LIN {X 0,Y 417.827,Z 989.103,A -85,B 0,C 180,E1 9549.226,E2 9549.226} C_VEL
LIN {X 0,Y 425.019,Z 968.051,A -85,B 0,C 180,E1 9548.696,E2 9548.696} C_VEL
LIN {X 0,Y 431.28,Z 946.58,A -85,B 0,C 180,E1 9548.255,E2 9548.255} C_VEL
LIN {X 0,Y 437.071,Z 922.468,A -85,B 0,C 180,E1 9547.851,E2 9547.851} C_VEL
LIN {X 0,Y 442.216,Z 893.072,A -85,B 0,C 180,E1 9547.412,E2 9547.412} C_VEL
LIN {X 0,Y 449.934,Z 826.101,A -85,B 0,C 180,E1 9546.506,E2 9546.506} C_VEL
LIN {X 0,Y 462.128,Z 717.477,A -85,B 0,C 180,E1 9545.058,E2 9545.058} C_VEL
LIN {X 0,Y 461.175,Z 715.537,A -85,B 0,C 180,E1 9543.107,E2 9543.107} C_VEL
LIN {X 0,Y 460.734,Z 712.812,A -85,B 0,C 180,E1 9540.249,E2 9540.249} C_VEL
LIN {X 0,Y 460.752,Z 712.952,A -85,B 0,C 180,E1 9538.881,E2 9538.881} C_VEL
LIN {X 0,Y 462.07,Z 717.316,A -85,B 0,C 180,E1 9534.54,E2 9534.54} C_VEL
LIN {X 0,Y 442.815,Z 887.011,A -85,B 0,C 180,E1 9532.28,E2 9532.28} C_VEL
LIN {X 0,Y 438.536,Z 912.989,A -85,B 0,C 180,E1 9531.901,E2 9531.901} C_VEL
LIN {X 0,Y 432.21,Z 940.386,A -85,B 0,C 180,E1 9531.4,E2 9531.4} C_VEL
LIN {X 0,Y 425.994,Z 962.099,A -85,B 0,C 180,E1 9530.901,E2 9530.901} C_VEL
LIN {X 0,Y 419.318,Z 981.985,A -85,B 0,C 180,E1 9530.35,E2 9530.35} C_VEL
LIN {X 0,Y 411.3,Z 1002.768,A -85,B 0,C 180,E1 9529.662,E2 9529.662} C_VEL
LIN {X 0,Y 400.652,Z 1026.921,A -85,B 0,C 180,E1 9528.701,E2 9528.701} C_VEL
LIN {X 0,Y 388.49,Z 1050.508,A -85,B 0,C 180,E1 9527.54,E2 9527.54} C_VEL
LIN {X 0,Y 377.454,Z 1069.69,A -85,B 0,C 180,E1 9526.414,E2 9526.414} C_VEL
LIN {X 0,Y 366.103,Z 1087.649,A -85,B 0,C 180,E1 9525.162,E2 9525.162} C_VEL
LIN {X 0,Y 352.977,Z 1106.617,A -85,B 0,C 180,E1 9523.599,E2 9523.599} C_VEL
LIN {X 0,Y 336.444,Z 1128.11,A -85,B 0,C 180,E1 9521.416,E2 9521.416} C_VEL
LIN {X 0,Y 323.396,Z 1143.609,A -85,B 0,C 180,E1 9519.493,E2 9519.493} C_VEL
LIN {X 0,Y 309.958,Z 1158.478,A -85,B 0,C 180,E1 9517.28,E2 9517.28} C_VEL
LIN {X 0,Y 296.26,Z 1172.662,A -85,B 0,C 180,E1 9514.73,E2 9514.73} C_VEL
LIN {X 0,Y 279.66,Z 1188.763,A -85,B 0,C 180,E1 9511.134,E2 9511.134} C_VEL
LIN {X 0,Y 264.844,Z 1202.074,A -85,B 0,C 180,E1 9507.319,E2 9507.319} C_VEL
LIN {X 0,Y 252.417,Z 1212.779,A -85,B 0,C 180,E1 9503.505,E2 9503.505} C_VEL
LIN {X 0,Y 241.138,Z 1222.219,A -85,B 0,C 180,E1 9499.339,E2 9499.339} C_VEL
LIN {X 0,Y 228.776,Z 1232.449,A -85,B 0,C 180,E1 9493.655,E2 9493.655} C_VEL
LIN {X 0,Y 218.042,Z 1241.237,A -85,B 0,C 180,E1 9487.067,E2 9487.067} C_VEL
LIN {X 0,Y 211.235,Z 1247.103,A -85,B 0,C 180,E1 9481.362,E2 9481.362} C_VEL
LIN {X 0,Y 206.073,Z 1251.951,A -85,B 0,C 180,E1 9475.261,E2 9475.261} C_VEL
LIN {X 0,Y 202.665,Z 1255.674,A -85,B 0,C 180,E1 9468.989,E2 9468.989} C_VEL
LIN {X 0,Y 200.676,Z 1258.635,A -85,B 0,C 180,E1 9461.774,E2 9461.774} C_VEL
LIN {X 0,Y 200.109,Z 1260.066,A -85,B 0,C 180,E1 9455.147,E2 9455.147} C_VEL
LIN {X 0,Y 200.012,Z 1260.414,A -85,B 0,C 180,E1 9449.414,E2 9449.414} C_VEL
LIN {X 0,Y 200.159,Z 1259.917,A -85,B 0,C 180,E1 9443.678,E2 9443.678} C_VEL
LIN {X 0,Y 200.883,Z 1258.243,A -85,B 0,C 180,E1 9437.044,E2 9437.044} C_VEL
LIN {X 0,Y 202.764,Z 1255.578,A -85,B 0,C 180,E1 9430.695,E2 9430.695} C_VEL
LIN {X 0,Y 206.041,Z 1252.022,A -85,B 0,C 180,E1 9424.707,E2 9424.707} C_VEL
LIN {X 0,Y 210.915,Z 1247.435,A -85,B 0,C 180,E1 9418.874,E2 9418.874} C_VEL
LIN {X 0,Y 217.804,Z 1241.484,A -85,B 0,C 180,E1 9413.016,E2 9413.016} C_VEL
LIN {X 0,Y 228.254,Z 1232.955,A -85,B 0,C 180,E1 9406.535,E2 9406.535} C_VEL
LIN {X 0,Y 240.93,Z 1222.476,A -85,B 0,C 180,E1 9400.66,E2 9400.66} C_VEL
LIN {X 0,Y 252.341,Z 1212.937,A -85,B 0,C 180,E1 9396.437,E2 9396.437} C_VEL
LIN {X 0,Y 264.769,Z 1202.248,A -85,B 0,C 180,E1 9392.619,E2 9392.619} C_VEL
LIN {X 0,Y 280.29,Z 1188.333,A -85,B 0,C 180,E1 9388.637,E2 9388.637} C_VEL
LIN {X 0,Y 296.47,Z 1172.615,A -85,B 0,C 180,E1 9385.148,E2 9385.148} C_VEL
LIN {X 0,Y 309.897,Z 1158.729,A -85,B 0,C 180,E1 9382.649,E2 9382.649} C_VEL
LIN {X 0,Y 323.344,Z 1143.878,A -85,B 0,C 180,E1 9380.436,E2 9380.436} C_VEL
LIN {X 0,Y 338.051,Z 1126.397,A -85,B 0,C 180,E1 9378.28,E2 9378.28} C_VEL
LIN {X 0,Y 354.452,Z 1104.814,A -85,B 0,C 180,E1 9376.136,E2 9376.136} C_VEL
LIN {X 0,Y 366.727,Z 1087.025,A -85,B 0,C 180,E1 9374.689,E2 9374.689} C_VEL
LIN {X 0,Y 377.843,Z 1069.412,A -85,B 0,C 180,E1 9373.467,E2 9373.467} C_VEL
LIN {X 0,Y 388.96,Z 1050.061,A -85,B 0,C 180,E1 9372.335,E2 9372.335} C_VEL
LIN {X 0,Y 401.541,Z 1025.448,A -85,B 0,C 180,E1 9371.137,E2 9371.137} C_VEL
LIN {X 0,Y 411.533,Z 1002.753,A -85,B 0,C 180,E1 9370.241,E2 9370.241} C_VEL
LIN {X 0,Y 419.451,Z 982.262,A -85,B 0,C 180,E1 9369.562,E2 9369.562} C_VEL
LIN {X 0,Y 426.457,Z 961.37,A -85,B 0,C 180,E1 9368.985,E2 9368.985} C_VEL
LIN {X 0,Y 433.115,Z 937.897,A -85,B 0,C 180,E1 9368.453,E2 9368.453} C_VEL
LIN {X 0,Y 439.471,Z 909.083,A -85,B 0,C 180,E1 9367.944,E2 9367.944} C_VEL
LIN {X 0,Y 443.203,Z 885.906,A -85,B 0,C 180,E1 9367.611,E2 9367.611} C_VEL
LIN {X 0,Y 461.965,Z 720.462,A -85,B 0,C 180,E1 9365.408,E2 9365.408} C_VEL
LIN {X 0,Y 462.048,Z 718.822,A -85,B 0,C 180,E1 9365.242,E2 9365.242} C_VEL
LIN {X 0,Y 461.875,Z 718.154,A -85,B 0,C 180,E1 9364.869,E2 9364.869} C_VEL
LIN {X 0,Y 461.404,Z 718.961,A -85,B 0,C 180,E1 9364.262,E2 9364.262} C_VEL
LIN {X 0,Y 460.384,Z 722.397,A -85,B 0,C 180,E1 9363.028,E2 9363.028} C_VEL
LIN {X 0,Y 460.143,Z 722.68,A -85,B 0,C 180,E1 9362.446,E2 9362.446} C_VEL
LIN {X 0,Y 460.028,Z 720.774,A -85,B 0,C 180,E1 9360.374,E2 9360.374} C_VEL
LIN {X 0,Y 460.024,Z 721.081,A -85,B 0,C 180,E1 9359.502,E2 9359.502} C_VEL
LIN {X 0,Y 460.881,Z 724.724,A -85,B 0,C 180,E1 9355.84,E2 9355.84} C_VEL
LIN {X 0,Y 441.798,Z 890.537,A -85,B 0,C 180,E1 9353.66,E2 9353.66} C_VEL
LIN {X 0,Y 437.471,Z 916.586,A -85,B 0,C 180,E1 9353.287,E2 9353.287} C_VEL
LIN {X 0,Y 430.938,Z 944.462,A -85,B 0,C 180,E1 9352.846,E2 9352.846} C_VEL
LIN {X 0,Y 424.579,Z 966.3,A -85,B 0,C 180,E1 9352.422,E2 9352.422} C_VEL
LIN {X 0,Y 417.486,Z 987.052,A -85,B 0,C 180,E1 9351.926,E2 9351.926} C_VEL
LIN {X 0,Y 409.171,Z 1008.194,A -85,B 0,C 180,E1 9351.313,E2 9351.313} C_VEL
LIN {X 0,Y 397.239,Z 1034.481,A -85,B 0,C 180,E1 9350.363,E2 9350.363} C_VEL
LIN {X 0,Y 385.977,Z 1055.977,A -85,B 0,C 180,E1 9349.401,E2 9349.401} C_VEL
LIN {X 0,Y 375.148,Z 1074.641,A -85,B 0,C 180,E1 9348.398,E2 9348.398} C_VEL
LIN {X 0,Y 363.473,Z 1092.965,A -85,B 0,C 180,E1 9347.232,E2 9347.232} C_VEL
LIN {X 0,Y 350.354,Z 1111.817,A -85,B 0,C 180,E1 9345.792,E2 9345.792} C_VEL
LIN {X 0,Y 332.937,Z 1134.393,A -85,B 0,C 180,E1 9343.661,E2 9343.661} C_VEL
LIN {X 0,Y 318.986,Z 1150.867,A -85,B 0,C 180,E1 9341.732,E2 9341.732} C_VEL
LIN {X 0,Y 305.166,Z 1166.066,A -85,B 0,C 180,E1 9339.584,E2 9339.584} C_VEL
LIN {X 0,Y 290.981,Z 1180.683,A -85,B 0,C 180,E1 9337.076,E2 9337.076} C_VEL
LIN {X 0,Y 273.041,Z 1197.971,A -85,B 0,C 180,E1 9333.336,E2 9333.336} C_VEL
LIN {X 0,Y 258.369,Z 1211.155,A -85,B 0,C 180,E1 9329.671,E2 9329.671} C_VEL
LIN {X 0,Y 245.406,Z 1222.365,A -85,B 0,C 180,E1 9325.787,E2 9325.787} C_VEL
LIN {X 0,Y 233.12,Z 1232.701,A -85,B 0,C 180,E1 9321.332,E2 9321.332} C_VEL
LIN {X 0,Y 219.784,Z 1243.853,A -85,B 0,C 180,E1 9315.157,E2 9315.157} C_VEL
LIN {X 0,Y 209.458,Z 1252.521,A -85,B 0,C 180,E1 9308.721,E2 9308.721} C_VEL
LIN {X 0,Y 202.639,Z 1258.658,A -85,B 0,C 180,E1 9302.886,E2 9302.886} C_VEL
LIN {X 0,Y 197.807,Z 1263.476,A -85,B 0,C 180,E1 9297.074,E2 9297.074} C_VEL
LIN {X 0,Y 194.579,Z 1267.316,A -85,B 0,C 180,E1 9291.096,E2 9291.096} C_VEL
LIN {X 0,Y 192.761,Z 1270.194,A -85,B 0,C 180,E1 9285.045,E2 9285.045} C_VEL
LIN {X 0,Y 192.092,Z 1271.973,A -85,B 0,C 180,E1 9279.602,E2 9279.602} C_VEL
LIN {X 0,Y 192.021,Z 1272.964,A -85,B 0,C 180,E1 9274.493,E2 9274.493} C_VEL
LIN {X 0,Y 192.011,Z 1273.253,A -85,B 0,C 180,E1 9269.119,E2 9269.119} C_VEL
LIN {X 0,Y 192.03,Z 1272.694,A -85,B 0,C 180,E1 9263.436,E2 9263.436} C_VEL
LIN {X 0,Y 192.495,Z 1270.789,A -85,B 0,C 180,E1 9256.497,E2 9256.497} C_VEL
LIN {X 0,Y 194.208,Z 1267.811,A -85,B 0,C 180,E1 9249.837,E2 9249.837} C_VEL
LIN {X 0,Y 197.39,Z 1263.897,A -85,B 0,C 180,E1 9243.544,E2 9243.544} C_VEL
LIN {X 0,Y 202.332,Z 1258.908,A -85,B 0,C 180,E1 9237.425,E2 9237.425} C_VEL
LIN {X 0,Y 209.057,Z 1252.815,A -85,B 0,C 180,E1 9231.573,E2 9231.573} C_VEL
LIN {X 0,Y 218.472,Z 1244.84,A -85,B 0,C 180,E1 9225.559,E2 9225.559} C_VEL
LIN {X 0,Y 232.595,Z 1233.068,A -85,B 0,C 180,E1 9218.876,E2 9218.876} C_VEL
LIN {X 0,Y 244.771,Z 1222.819,A -85,B 0,C 180,E1 9214.418,E2 9214.418} C_VEL
LIN {X 0,Y 257.409,Z 1211.888,A -85,B 0,C 180,E1 9210.588,E2 9210.588} C_VEL
LIN {X 0,Y 271.526,Z 1199.21,A -85,B 0,C 180,E1 9207.009,E2 9207.009} C_VEL
LIN {X 0,Y 290.131,Z 1181.388,A -85,B 0,C 180,E1 9203.08,E2 9203.08} C_VEL
LIN {X 0,Y 304.281,Z 1166.834,A -85,B 0,C 180,E1 9200.557,E2 9200.557} C_VEL
LIN {X 0,Y 317.858,Z 1151.944,A -85,B 0,C 180,E1 9198.427,E2 9198.427} C_VEL
LIN {X 0,Y 330.96,Z 1136.545,A -85,B 0,C 180,E1 9196.587,E2 9196.587} C_VEL
LIN {X 0,Y 345.571,Z 1118.021,A -85,B 0,C 180,E1 9194.751,E2 9194.751} C_VEL
LIN {X 0,Y 361.758,Z 1095.238,A -85,B 0,C 180,E1 9192.937,E2 9192.937} C_VEL
LIN {X 0,Y 374.151,Z 1075.917,A -85,B 0,C 180,E1 9191.688,E2 9191.688} C_VEL
LIN {X 0,Y 385.049,Z 1057.238,A -85,B 0,C 180,E1 9190.671,E2 9190.671} C_VEL
LIN {X 0,Y 396.029,Z 1036.414,A -85,B 0,C 180,E1 9189.725,E2 9189.725} C_VEL
LIN {X 0,Y 408.494,Z 1009.289,A -85,B 0,C 180,E1 9188.729,E2 9188.729} C_VEL
LIN {X 0,Y 417.04,Z 987.634,A -85,B 0,C 180,E1 9188.096,E2 9188.096} C_VEL
LIN {X 0,Y 424.156,Z 966.885,A -85,B 0,C 180,E1 9187.597,E2 9187.597} C_VEL
LIN {X 0,Y 430.377,Z 945.642,A -85,B 0,C 180,E1 9187.18,E2 9187.18} C_VEL
LIN {X 0,Y 436.755,Z 919.053,A -85,B 0,C 180,E1 9186.754,E2 9186.754} C_VEL
LIN {X 0,Y 441.451,Z 891.288,A -85,B 0,C 180,E1 9186.354,E2 9186.354} C_VEL
LIN {X 0,Y 454.023,Z 782.367,A -85,B 0,C 180,E1 9184.916,E2 9184.916} C_VEL
LIN {X 0,Y 460.65,Z 724.372,A -85,B 0,C 180,E1 9184.139,E2 9184.139} C_VEL
LIN {X 0,Y 459.759,Z 720.752,A -85,B 0,C 180,E1 9180.249,E2 9180.249} C_VEL
LIN {X 0,Y 459.767,Z 720.977,A -85,B 0,C 180,E1 9178.878,E2 9178.878} C_VEL
LIN {X 0,Y 460.589,Z 724.432,A -85,B 0,C 180,E1 9175.442,E2 9175.442} C_VEL
LIN {X 0,Y 441.811,Z 887.296,A -85,B 0,C 180,E1 9173.309,E2 9173.309} C_VEL
LIN {X 0,Y 437.45,Z 913.431,A -85,B 0,C 180,E1 9172.937,E2 9172.937} C_VEL
LIN {X 0,Y 431.084,Z 940.66,A -85,B 0,C 180,E1 9172.454,E2 9172.454} C_VEL
LIN {X 0,Y 424.797,Z 962.372,A -85,B 0,C 180,E1 9171.971,E2 9171.971} C_VEL
LIN {X 0,Y 418.044,Z 982.258,A -85,B 0,C 180,E1 9171.437,E2 9171.437} C_VEL
LIN {X 0,Y 410.172,Z 1002.448,A -85,B 0,C 180,E1 9170.791,E2 9170.791} C_VEL
LIN {X 0,Y 399.603,Z 1026.198,A -85,B 0,C 180,E1 9169.881,E2 9169.881} C_VEL
LIN {X 0,Y 387.316,Z 1049.895,A -85,B 0,C 180,E1 9168.762,E2 9168.762} C_VEL
LIN {X 0,Y 376.073,Z 1069.234,A -85,B 0,C 180,E1 9167.665,E2 9167.665} C_VEL
LIN {X 0,Y 364.98,Z 1086.599,A -85,B 0,C 180,E1 9166.499,E2 9166.499} C_VEL
LIN {X 0,Y 352.723,Z 1104.142,A -85,B 0,C 180,E1 9165.121,E2 9165.121} C_VEL
LIN {X 0,Y 336.944,Z 1124.789,A -85,B 0,C 180,E1 9163.157,E2 9163.157} C_VEL
LIN {X 0,Y 320.707,Z 1143.762,A -85,B 0,C 180,E1 9160.891,E2 9160.891} C_VEL
LIN {X 0,Y 307.656,Z 1157.92,A -85,B 0,C 180,E1 9158.836,E2 9158.836} C_VEL
LIN {X 0,Y 294.353,Z 1171.42,A -85,B 0,C 180,E1 9156.485,E2 9156.485} C_VEL
LIN {X 0,Y 280.096,Z 1184.997,A -85,B 0,C 180,E1 9153.612,E2 9153.612} C_VEL
LIN {X 0,Y 262.461,Z 1200.665,A -85,B 0,C 180,E1 9149.402,E2 9149.402} C_VEL
LIN {X 0,Y 248.783,Z 1212.049,A -85,B 0,C 180,E1 9145.456,E2 9145.456} C_VEL
LIN {X 0,Y 236.897,Z 1221.601,A -85,B 0,C 180,E1 9141.316,E2 9141.316} C_VEL
LIN {X 0,Y 225.735,Z 1230.361,A -85,B 0,C 180,E1 9136.568,E2 9136.568} C_VEL
LIN {X 0,Y 214.002,Z 1239.604,A -85,B 0,C 180,E1 9130.131,E2 9130.131} C_VEL
LIN {X 0,Y 204.797,Z 1246.886,A -85,B 0,C 180,E1 9123.132,E2 9123.132} C_VEL
LIN {X 0,Y 199.289,Z 1251.628,A -85,B 0,C 180,E1 9117.15,E2 9117.15} C_VEL
LIN {X 0,Y 195.512,Z 1255.333,A -85,B 0,C 180,E1 9110.961,E2 9110.961} C_VEL
LIN {X 0,Y 193.263,Z 1258.045,A -85,B 0,C 180,E1 9104.65,E2 9104.65} C_VEL
LIN {X 0,Y 192.325,Z 1259.643,A -85,B 0,C 180,E1 9098.957,E2 9098.957} C_VEL
LIN {X 0,Y 192.078,Z 1260.431,A -85,B 0,C 180,E1 9093.866,E2 9093.866} C_VEL
LIN {X 0,Y 192.041,Z 1260.588,A -85,B 0,C 180,E1 9088.196,E2 9088.196} C_VEL
LIN {X 0,Y 192.229,Z 1259.986,A -85,B 0,C 180,E1 9082.515,E2 9082.515} C_VEL
LIN {X 0,Y 193.113,Z 1258.293,A -85,B 0,C 180,E1 9075.902,E2 9075.902} C_VEL
LIN {X 0,Y 195.206,Z 1255.694,A -85,B 0,C 180,E1 9069.603,E2 9069.603} C_VEL
LIN {X 0,Y 198.826,Z 1252.094,A -85,B 0,C 180,E1 9063.399,E2 9063.399} C_VEL
LIN {X 0,Y 204.155,Z 1247.461,A -85,B 0,C 180,E1 9057.389,E2 9057.389} C_VEL
LIN {X 0,Y 211.593,Z 1241.465,A -85,B 0,C 180,E1 9051.395,E2 9051.395} C_VEL
LIN {X 0,Y 223.228,Z 1232.464,A -85,B 0,C 180,E1 9044.573,E2 9044.573} C_VEL
LIN {X 0,Y 235.705,Z 1222.638,A -85,B 0,C 180,E1 9039.063,E2 9039.063} C_VEL
LIN {X 0,Y 247.471,Z 1213.209,A -85,B 0,C 180,E1 9034.881,E2 9034.881} C_VEL
LIN {X 0,Y 260.366,Z 1202.52,A -85,B 0,C 180,E1 9031.072,E2 9031.072} C_VEL
LIN {X 0,Y 276.441,Z 1188.567,A -85,B 0,C 180,E1 9027.113,E2 9027.113} C_VEL
LIN {X 0,Y 292.76,Z 1173.164,A -85,B 0,C 180,E1 9023.734,E2 9023.734} C_VEL
LIN {X 0,Y 306.964,Z 1158.832,A -85,B 0,C 180,E1 9021.197,E2 9021.197} C_VEL
LIN {X 0,Y 320.554,Z 1144.146,A -85,B 0,C 180,E1 9019.052,E2 9019.052} C_VEL
LIN {X 0,Y 335.56,Z 1126.664,A -85,B 0,C 180,E1 9016.945,E2 9016.945} C_VEL
LIN {X 0,Y 352.261,Z 1105.079,A -85,B 0,C 180,E1 9014.855,E2 9014.855} C_VEL
LIN {X 0,Y 364.365,Z 1087.854,A -85,B 0,C 180,E1 9013.489,E2 9013.489} C_VEL
LIN {X 0,Y 375.704,Z 1070.206,A -85,B 0,C 180,E1 9012.293,E2 9012.293} C_VEL
LIN {X 0,Y 386.898,Z 1051.047,A -85,B 0,C 180,E1 9011.199,E2 9011.199} C_VEL
LIN {X 0,Y 399.143,Z 1027.673,A -85,B 0,C 180,E1 9010.083,E2 9010.083} C_VEL
LIN {X 0,Y 410.175,Z 1003.011,A -85,B 0,C 180,E1 9009.132,E2 9009.132} C_VEL
LIN {X 0,Y 418.052,Z 982.895,A -85,B 0,C 180,E1 9008.486,E2 9008.486} C_VEL
LIN {X 0,Y 425.043,Z 962.361,A -85,B 0,C 180,E1 9007.934,E2 9007.934} C_VEL
LIN {X 0,Y 431.436,Z 940.255,A -85,B 0,C 180,E1 9007.442,E2 9007.442} C_VEL
LIN {X 0,Y 437.93,Z 912.126,A -85,B 0,C 180,E1 9006.948,E2 9006.948} C_VEL
LIN {X 0,Y 442.084,Z 887.108,A -85,B 0,C 180,E1 9006.595,E2 9006.595} C_VEL
LIN {X 0,Y 460.841,Z 724.411,A -85,B 0,C 180,E1 9004.449,E2 9004.449} C_VEL
LIN {X 0,Y 460.143,Z 722.68,A -85,B 0,C 180,E1 9002.446,E2 9002.446} C_VEL
LIN {X 0,Y 459.896,Z 722.863,A -85,B 0,C 180,E1 9001.548,E2 9001.548} C_VEL
LIN {X 0,Y 459.438,Z 725.568,A -85,B 0,C 180,E1 9000.265,E2 9000.265} C_VEL
LIN {X 0,Y 459.096,Z 730.018,A -85,B 0,C 180,E1 8998.499,E2 8998.499} C_VEL
LIN {X 0,Y 459.139,Z 730.581,A -85,B 0,C 180,E1 8998.079,E2 8998.079} C_VEL
LIN {X 0,Y 459.5,Z 731.895,A -85,B 0,C 180,E1 8996.745,E2 8996.745} C_VEL
LIN {X 0,Y 440.967,Z 890.402,A -85,B 0,C 180,E1 8994.699,E2 8994.699} C_VEL
LIN {X 0,Y 436.485,Z 916.989,A -85,B 0,C 180,E1 8994.327,E2 8994.327} C_VEL
LIN {X 0,Y 429.907,Z 944.576,A -85,B 0,C 180,E1 8993.905,E2 8993.905} C_VEL
LIN {X 0,Y 423.688,Z 965.735,A -85,B 0,C 180,E1 8993.511,E2 8993.511} C_VEL
LIN {X 0,Y 416.548,Z 986.465,A -85,B 0,C 180,E1 8993.037,E2 8993.037} C_VEL
LIN {X 0,Y 408.159,Z 1007.61,A -85,B 0,C 180,E1 8992.45,E2 8992.45} C_VEL
LIN {X 0,Y 396.28,Z 1033.592,A -85,B 0,C 180,E1 8991.551,E2 8991.551} C_VEL
LIN {X 0,Y 384.638,Z 1055.568,A -85,B 0,C 180,E1 8990.607,E2 8990.607} C_VEL
LIN {X 0,Y 373.581,Z 1074.375,A -85,B 0,C 180,E1 8989.633,E2 8989.633} C_VEL
LIN {X 0,Y 361.975,Z 1092.352,A -85,B 0,C 180,E1 8988.528,E2 8988.528} C_VEL
LIN {X 0,Y 349.171,Z 1110.504,A -85,B 0,C 180,E1 8987.195,E2 8987.195} C_VEL
LIN {X 0,Y 332.606,Z 1131.868,A -85,B 0,C 180,E1 8985.28,E2 8985.28} C_VEL
LIN {X 0,Y 316.811,Z 1150.212,A -85,B 0,C 180,E1 8983.218,E2 8983.218} C_VEL
LIN {X 0,Y 303.164,Z 1164.936,A -85,B 0,C 180,E1 8981.204,E2 8981.204} C_VEL
LIN {X 0,Y 289.398,Z 1178.844,A -85,B 0,C 180,E1 8978.903,E2 8978.903} C_VEL
LIN {X 0,Y 274.618,Z 1192.874,A -85,B 0,C 180,E1 8976.065,E2 8976.065} C_VEL
LIN {X 0,Y 255.602,Z 1209.708,A -85,B 0,C 180,E1 8971.679,E2 8971.679} C_VEL
LIN {X 0,Y 241.438,Z 1221.524,A -85,B 0,C 180,E1 8967.67,E2 8967.67} C_VEL
LIN {X 0,Y 229.094,Z 1231.483,A -85,B 0,C 180,E1 8963.439,E2 8963.439} C_VEL
LIN {X 0,Y 216.998,Z 1241.082,A -85,B 0,C 180,E1 8958.3,E2 8958.3} C_VEL
LIN {X 0,Y 204.163,Z 1251.305,A -85,B 0,C 180,E1 8951.03,E2 8951.03} C_VEL
LIN {X 0,Y 195.973,Z 1258.119,A -85,B 0,C 180,E1 8944.509,E2 8944.509} C_VEL
LIN {X 0,Y 190.446,Z 1263.204,A -85,B 0,C 180,E1 8938.212,E2 8938.212} C_VEL
LIN {X 0,Y 186.902,Z 1267.045,A -85,B 0,C 180,E1 8932.006,E2 8932.006} C_VEL
LIN {X 0,Y 184.877,Z 1269.927,A -85,B 0,C 180,E1 8925.699,E2 8925.699} C_VEL
LIN {X 0,Y 184.111,Z 1271.707,A -85,B 0,C 180,E1 8920.022,E2 8920.022} C_VEL
LIN {X 0,Y 184.023,Z 1272.7,A -85,B 0,C 180,E1 8914.689,E2 8914.689} C_VEL
LIN {X 0,Y 184.016,Z 1272.99,A -85,B 0,C 180,E1 8909.08,E2 8909.08} C_VEL
LIN {X 0,Y 184.032,Z 1272.502,A -85,B 0,C 180,E1 8903.463,E2 8903.463} C_VEL
LIN {X 0,Y 184.528,Z 1270.641,A -85,B 0,C 180,E1 8896.222,E2 8896.222} C_VEL
LIN {X 0,Y 186.493,Z 1267.54,A -85,B 0,C 180,E1 8888.964,E2 8888.964} C_VEL
LIN {X 0,Y 189.989,Z 1263.624,A -85,B 0,C 180,E1 8882.428,E2 8882.428} C_VEL
LIN {X 0,Y 195.332,Z 1258.633,A -85,B 0,C 180,E1 8876.103,E2 8876.103} C_VEL
LIN {X 0,Y 202.534,Z 1252.538,A -85,B 0,C 180,E1 8870.094,E2 8870.094} C_VEL
LIN {X 0,Y 212.503,Z 1244.576,A -85,B 0,C 180,E1 8863.974,E2 8863.974} C_VEL
LIN {X 0,Y 227.297,Z 1232.862,A -85,B 0,C 180,E1 8857.252,E2 8857.252} C_VEL
LIN {X 0,Y 240.09,Z 1222.54,A -85,B 0,C 180,E1 8852.752,E2 8852.752} C_VEL
LIN {X 0,Y 252.745,Z 1212.003,A -85,B 0,C 180,E1 8849.065,E2 8849.065} C_VEL
LIN {X 0,Y 267.058,Z 1199.578,A -85,B 0,C 180,E1 8845.564,E2 8845.564} C_VEL
LIN {X 0,Y 284.582,Z 1183.459,A -85,B 0,C 180,E1 8841.973,E2 8841.973} C_VEL
LIN {X 0,Y 301.437,Z 1166.556,A -85,B 0,C 180,E1 8839.063,E2 8839.063} C_VEL
LIN {X 0,Y 314.76,Z 1152.284,A -85,B 0,C 180,E1 8837.064,E2 8837.064} C_VEL
LIN {X 0,Y 327.944,Z 1137.144,A -85,B 0,C 180,E1 8835.29,E2 8835.29} C_VEL
LIN {X 0,Y 341.532,Z 1120.308,A -85,B 0,C 180,E1 8833.642,E2 8833.642} C_VEL
LIN {X 0,Y 357.586,Z 1098.576,A -85,B 0,C 180,E1 8831.905,E2 8831.905} C_VEL
LIN {X 0,Y 371.566,Z 1077.273,A -85,B 0,C 180,E1 8830.544,E2 8830.544} C_VEL
LIN {X 0,Y 382.691,Z 1058.599,A -85,B 0,C 180,E1 8829.548,E2 8829.548} C_VEL
LIN {X 0,Y 392.911,Z 1039.674,A -85,B 0,C 180,E1 8828.701,E2 8828.701} C_VEL
LIN {X 0,Y 402.747,Z 1019.375,A -85,B 0,C 180,E1 8827.94,E2 8827.94} C_VEL
LIN {X 0,Y 413.608,Z 993.813,A -85,B 0,C 180,E1 8827.157,E2 8827.157} C_VEL
LIN {X 0,Y 422.401,Z 968.987,A -85,B 0,C 180,E1 8826.563,E2 8826.563} C_VEL
LIN {X 0,Y 428.782,Z 947.773,A -85,B 0,C 180,E1 8826.155,E2 8826.155} C_VEL
LIN {X 0,Y 434.273,Z 925.807,A -85,B 0,C 180,E1 8825.807,E2 8825.807} C_VEL
LIN {X 0,Y 439.562,Z 898.725,A -85,B 0,C 180,E1 8825.417,E2 8825.417} C_VEL
LIN {X 0,Y 444.883,Z 856.168,A -85,B 0,C 180,E1 8824.857,E2 8824.857} C_VEL
LIN {X 0,Y 459.264,Z 731.613,A -85,B 0,C 180,E1 8823.245,E2 8823.245} C_VEL
LIN {X 0,Y 458.776,Z 728.693,A -85,B 0,C 180,E1 8820.125,E2 8820.125} C_VEL
LIN {X 0,Y 458.785,Z 728.857,A -85,B 0,C 180,E1 8819.001,E2 8819.001} C_VEL
LIN {X 0,Y 459.218,Z 731.591,A -85,B 0,C 180,E1 8816.349,E2 8816.349} C_VEL
LIN {X 0,Y 440.936,Z 887.687,A -85,B 0,C 180,E1 8814.34,E2 8814.34} C_VEL
LIN {X 0,Y 436.42,Z 914.357,A -85,B 0,C 180,E1 8813.97,E2 8813.97} C_VEL
LIN {X 0,Y 430.016,Z 941.258,A -85,B 0,C 180,E1 8813.506,E2 8813.506} C_VEL
LIN {X 0,Y 423.75,Z 962.645,A -85,B 0,C 180,E1 8813.046,E2 8813.046} C_VEL
LIN {X 0,Y 416.922,Z 982.53,A -85,B 0,C 180,E1 8812.531,E2 8812.531} C_VEL
LIN {X 0,Y 408.693,Z 1003.361,A -85,B 0,C 180,E1 8811.885,E2 8811.885} C_VEL
LIN {X 0,Y 397.336,Z 1028.387,A -85,B 0,C 180,E1 8810.948,E2 8810.948} C_VEL
LIN {X 0,Y 385.358,Z 1050.971,A -85,B 0,C 180,E1 8809.903,E2 8809.903} C_VEL
LIN {X 0,Y 373.966,Z 1070.234,A -85,B 0,C 180,E1 8808.838,E2 8808.838} C_VEL
LIN {X 0,Y 362.266,Z 1088.194,A -85,B 0,C 180,E1 8807.658,E2 8807.658} C_VEL
LIN {X 0,Y 348.513,Z 1107.423,A -85,B 0,C 180,E1 8806.162,E2 8806.162} C_VEL
LIN {X 0,Y 331.564,Z 1128.657,A -85,B 0,C 180,E1 8804.113,E2 8804.113} C_VEL
LIN {X 0,Y 317.543,Z 1144.645,A -85,B 0,C 180,E1 8802.215,E2 8802.215} C_VEL
LIN {X 0,Y 303.954,Z 1159.027,A -85,B 0,C 180,E1 8800.156,E2 8800.156} C_VEL
LIN {X 0,Y 289.572,Z 1173.211,A -85,B 0,C 180,E1 8797.697,E2 8797.697} C_VEL
LIN {X 0,Y 272.019,Z 1189.313,A -85,B 0,C 180,E1 8794.204,E2 8794.204} C_VEL
LIN {X 0,Y 256.226,Z 1202.625,A -85,B 0,C 180,E1 8790.459,E2 8790.459} C_VEL
LIN {X 0,Y 242.859,Z 1213.33,A -85,B 0,C 180,E1 8786.673,E2 8786.673} C_VEL
LIN {X 0,Y 230.598,Z 1222.771,A -85,B 0,C 180,E1 8782.491,E2 8782.491} C_VEL
LIN {X 0,Y 217.021,Z 1232.999,A -85,B 0,C 180,E1 8776.694,E2 8776.694} C_VEL
LIN {X 0,Y 205.214,Z 1241.637,A -85,B 0,C 180,E1 8770.008,E2 8770.008} C_VEL
LIN {X 0,Y 197.265,Z 1247.649,A -85,B 0,C 180,E1 8763.869,E2 8763.869} C_VEL
LIN {X 0,Y 191.518,Z 1252.295,A -85,B 0,C 180,E1 8757.671,E2 8757.671} C_VEL
LIN {X 0,Y 187.493,Z 1255.998,A -85,B 0,C 180,E1 8751.049,E2 8751.049} C_VEL
LIN {X 0,Y 185.052,Z 1258.843,A -85,B 0,C 180,E1 8743.738,E2 8743.738} C_VEL
LIN {X 0,Y 184.167,Z 1260.545,A -85,B 0,C 180,E1 8736.219,E2 8736.219} C_VEL
LIN {X 0,Y 184.035,Z 1260.972,A -85,B 0,C 180,E1 8729.986,E2 8729.986} C_VEL
LIN {X 0,Y 184.166,Z 1260.559,A -85,B 0,C 180,E1 8723.752,E2 8723.752} C_VEL
LIN {X 0,Y 184.974,Z 1258.99,A -85,B 0,C 180,E1 8716.546,E2 8716.546} C_VEL
LIN {X 0,Y 187.425,Z 1256.096,A -85,B 0,C 180,E1 8709.005,E2 8709.005} C_VEL
LIN {X 0,Y 191.256,Z 1252.562,A -85,B 0,C 180,E1 8702.595,E2 8702.595} C_VEL
LIN {X 0,Y 196.908,Z 1247.977,A -85,B 0,C 180,E1 8696.379,E2 8696.379} C_VEL
LIN {X 0,Y 204.354,Z 1242.323,A -85,B 0,C 180,E1 8690.486,E2 8690.486} C_VEL
LIN {X 0,Y 214.479,Z 1234.87,A -85,B 0,C 180,E1 8684.484,E2 8684.484} C_VEL
LIN {X 0,Y 229.374,Z 1223.806,A -85,B 0,C 180,E1 8677.892,E2 8677.892} C_VEL
LIN {X 0,Y 242.153,Z 1213.985,A -85,B 0,C 180,E1 8673.464,E2 8673.464} C_VEL
LIN {X 0,Y 254.78,Z 1203.915,A -85,B 0,C 180,E1 8669.837,E2 8669.837} C_VEL
LIN {X 0,Y 268.272,Z 1192.614,A -85,B 0,C 180,E1 8666.539,E2 8666.539} C_VEL
LIN {X 0,Y 284.845,Z 1177.905,A -85,B 0,C 180,E1 8663.103,E2 8663.103} C_VEL
LIN {X 0,Y 302.283,Z 1160.933,A -85,B 0,C 180,E1 8660.031,E2 8660.031} C_VEL
LIN {X 0,Y 316.618,Z 1145.873,A -85,B 0,C 180,E1 8657.838,E2 8657.838} C_VEL
LIN {X 0,Y 330.062,Z 1130.654,A -85,B 0,C 180,E1 8656.002,E2 8656.002} C_VEL
LIN {X 0,Y 343.727,Z 1113.907,A -85,B 0,C 180,E1 8654.316,E2 8654.316} C_VEL
LIN {X 0,Y 360.466,Z 1091.197,A -85,B 0,C 180,E1 8652.453,E2 8652.453} C_VEL
LIN {X 0,Y 373.053,Z 1072.08,A -85,B 0,C 180,E1 8651.172,E2 8651.172} C_VEL
LIN {X 0,Y 383.984,Z 1053.804,A -85,B 0,C 180,E1 8650.145,E2 8650.145} C_VEL
LIN {X 0,Y 394.099,Z 1035.09,A -85,B 0,C 180,E1 8649.245,E2 8649.245} C_VEL
LIN {X 0,Y 404.352,Z 1013.889,A -85,B 0,C 180,E1 8648.389,E2 8648.389} C_VEL
LIN {X 0,Y 415.532,Z 986.984,A -85,B 0,C 180,E1 8647.502,E2 8647.502} C_VEL
LIN {X 0,Y 423.164,Z 965.251,A -85,B 0,C 180,E1 8646.921,E2 8646.921} C_VEL
LIN {X 0,Y 429.536,Z 943.912,A -85,B 0,C 180,E1 8646.45,E2 8646.45} C_VEL
LIN {X 0,Y 434.932,Z 922.131,A -85,B 0,C 180,E1 8646.058,E2 8646.058} C_VEL
LIN {X 0,Y 440.241,Z 894.612,A -85,B 0,C 180,E1 8645.658,E2 8645.658} C_VEL
LIN {X 0,Y 445.831,Z 849.431,A -85,B 0,C 180,E1 8645.066,E2 8645.066} C_VEL
LIN {X 0,Y 459.464,Z 731.631,A -85,B 0,C 180,E1 8643.528,E2 8643.528} C_VEL
LIN {X 0,Y 459.053,Z 728.715,A -85,B 0,C 180,E1 8640.374,E2 8640.374} C_VEL
LIN {X 0,Y 459.039,Z 729.1,A -85,B 0,C 180,E1 8639.501,E2 8639.501} C_VEL
LIN {X 0,Y 459.139,Z 730.581,A -85,B 0,C 180,E1 8638.079,E2 8638.079} C_VEL
LIN {X 0,Y 459.083,Z 731.777,A -85,B 0,C 180,E1 8637.795,E2 8637.795} C_VEL
LIN {X 0,Y 458.811,Z 734.647,A -85,B 0,C 180,E1 8637.566,E2 8637.566} C_VEL
LIN {X 0,Y 458.243,Z 739.648,A -85,B 0,C 180,E1 8637.441,E2 8637.441} C_VEL
LIN {X 0,Y 456.477,Z 753.93,A -85,B 0,C 180,E1 8637.469,E2 8637.469} C_VEL
LIN {X 0,Y 440.281,Z 890.266,A -85,B 0,C 180,E1 8635.741,E2 8635.741} C_VEL
LIN {X 0,Y 435.647,Z 917.368,A -85,B 0,C 180,E1 8635.372,E2 8635.372} C_VEL
LIN {X 0,Y 429.042,Z 944.627,A -85,B 0,C 180,E1 8634.97,E2 8634.97} C_VEL
LIN {X 0,Y 422.852,Z 965.479,A -85,B 0,C 180,E1 8634.598,E2 8634.598} C_VEL
LIN {X 0,Y 415.644,Z 986.207,A -85,B 0,C 180,E1 8634.144,E2 8634.144} C_VEL
LIN {X 0,Y 407.188,Z 1007.312,A -85,B 0,C 180,E1 8633.583,E2 8633.583} C_VEL
LIN {X 0,Y 395.369,Z 1032.939,A -85,B 0,C 180,E1 8632.735,E2 8632.735} C_VEL
LIN {X 0,Y 383.431,Z 1055.23,A -85,B 0,C 180,E1 8631.817,E2 8631.817} C_VEL
LIN {X 0,Y 372.222,Z 1074.059,A -85,B 0,C 180,E1 8630.881,E2 8630.881} C_VEL
LIN {X 0,Y 360.144,Z 1092.5,A -85,B 0,C 180,E1 8629.785,E2 8629.785} C_VEL
LIN {X 0,Y 346.979,Z 1110.851,A -85,B 0,C 180,E1 8628.479,E2 8628.479} C_VEL
LIN {X 0,Y 329.086,Z 1133.341,A -85,B 0,C 180,E1 8626.499,E2 8626.499} C_VEL
LIN {X 0,Y 314.22,Z 1150.245,A -85,B 0,C 180,E1 8624.639,E2 8624.639} C_VEL
LIN {X 0,Y 299.729,Z 1165.521,A -85,B 0,C 180,E1 8622.589,E2 8622.589} C_VEL
LIN {X 0,Y 284.855,Z 1180.136,A -85,B 0,C 180,E1 8620.191,E2 8620.191} C_VEL
LIN {X 0,Y 265.891,Z 1197.421,A -85,B 0,C 180,E1 8616.59,E2 8616.59} C_VEL
LIN {X 0,Y 250.256,Z 1210.603,A -85,B 0,C 180,E1 8613.014,E2 8613.014} C_VEL
LIN {X 0,Y 236.349,Z 1221.775,A -85,B 0,C 180,E1 8609.198,E2 8609.198} C_VEL
LIN {X 0,Y 222.939,Z 1232.148,A -85,B 0,C 180,E1 8604.729,E2 8604.729} C_VEL
LIN {X 0,Y 208.304,Z 1243.234,A -85,B 0,C 180,E1 8598.504,E2 8598.504} C_VEL
LIN {X 0,Y 196.615,Z 1251.971,A -85,B 0,C 180,E1 8591.789,E2 8591.789} C_VEL
LIN {X 0,Y 188.802,Z 1258.11,A -85,B 0,C 180,E1 8585.645,E2 8585.645} C_VEL
LIN {X 0,Y 182.923,Z 1263.147,A -85,B 0,C 180,E1 8579.125,E2 8579.125} C_VEL
LIN {X 0,Y 178.974,Z 1267.111,A -85,B 0,C 180,E1 8572.342,E2 8572.342} C_VEL
LIN {X 0,Y 176.806,Z 1270.019,A -85,B 0,C 180,E1 8565.429,E2 8565.429} C_VEL
LIN {X 0,Y 176.071,Z 1271.807,A -85,B 0,C 180,E1 8558.835,E2 8558.835} C_VEL
LIN {X 0,Y 176.031,Z 1272.538,A -85,B 0,C 180,E1 8553.597,E2 8553.597} C_VEL
LIN {X 0,Y 176.034,Z 1272.681,A -85,B 0,C 180,E1 8548.388,E2 8548.388} C_VEL
LIN {X 0,Y 176.04,Z 1272.093,A -85,B 0,C 180,E1 8542.509,E2 8542.509} C_VEL
LIN {X 0,Y 176.678,Z 1270.253,A -85,B 0,C 180,E1 8535.262,E2 8535.262} C_VEL
LIN {X 0,Y 178.822,Z 1267.269,A -85,B 0,C 180,E1 8528.016,E2 8528.016} C_VEL
LIN {X 0,Y 182.767,Z 1263.258,A -85,B 0,C 180,E1 8521.085,E2 8521.085} C_VEL
LIN {X 0,Y 188.769,Z 1258.093,A -85,B 0,C 180,E1 8514.382,E2 8514.382} C_VEL
LIN {X 0,Y 196.995,Z 1251.633,A -85,B 0,C 180,E1 8507.954,E2 8507.954} C_VEL
LIN {X 0,Y 209.83,Z 1242.014,A -85,B 0,C 180,E1 8500.756,E2 8500.756} C_VEL
LIN {X 0,Y 223.483,Z 1231.641,A -85,B 0,C 180,E1 8495.064,E2 8495.064} C_VEL
LIN {X 0,Y 236.383,Z 1221.652,A -85,B 0,C 180,E1 8490.786,E2 8490.786} C_VEL
LIN {X 0,Y 250.181,Z 1210.552,A -85,B 0,C 180,E1 8486.998,E2 8486.998} C_VEL
LIN {X 0,Y 267.352,Z 1196.061,A -85,B 0,C 180,E1 8483.102,E2 8483.102} C_VEL
LIN {X 0,Y 284.77,Z 1180.048,A -85,B 0,C 180,E1 8479.815,E2 8479.815} C_VEL
LIN {X 0,Y 299.642,Z 1165.42,A -85,B 0,C 180,E1 8477.416,E2 8477.416} C_VEL
LIN {X 0,Y 314.13,Z 1150.13,A -85,B 0,C 180,E1 8475.365,E2 8475.365} C_VEL
LIN {X 0,Y 329.437,Z 1132.697,A -85,B 0,C 180,E1 8473.451,E2 8473.451} C_VEL
LIN {X 0,Y 346.886,Z 1110.681,A -85,B 0,C 180,E1 8471.521,E2 8471.521} C_VEL
LIN {X 0,Y 360.05,Z 1092.303,A -85,B 0,C 180,E1 8470.214,E2 8470.214} C_VEL
LIN {X 0,Y 372.049,Z 1073.96,A -85,B 0,C 180,E1 8469.124,E2 8469.124} C_VEL
LIN {X 0,Y 383.763,Z 1054.24,A -85,B 0,C 180,E1 8468.147,E2 8468.147} C_VEL
LIN {X 0,Y 396.962,Z 1029.21,A -85,B 0,C 180,E1 8467.135,E2 8467.135} C_VEL
LIN {X 0,Y 407.417,Z 1006.189,A -85,B 0,C 180,E1 8466.391,E2 8466.391} C_VEL
LIN {X 0,Y 415.549,Z 985.796,A -85,B 0,C 180,E1 8465.851,E2 8465.851} C_VEL
LIN {X 0,Y 422.757,Z 965,A -85,B 0,C 180,E1 8465.396,E2 8465.396} C_VEL
LIN {X 0,Y 429.693,Z 941.377,A -85,B 0,C 180,E1 8464.982,E2 8464.982} C_VEL
LIN {X 0,Y 436.354,Z 912.131,A -85,B 0,C 180,E1 8464.558,E2 8464.558} C_VEL
LIN {X 0,Y 440.212,Z 888.888,A -85,B 0,C 180,E1 8464.244,E2 8464.244} C_VEL
LIN {X 0,Y 457.991,Z 738.796,A -85,B 0,C 180,E1 8462.33,E2 8462.33} C_VEL
LIN {X 0,Y 457.801,Z 736.634,A -85,B 0,C 180,E1 8460.125,E2 8460.125} C_VEL
LIN {X 0,Y 457.8,Z 736.878,A -85,B 0,C 180,E1 8458.999,E2 8458.999} C_VEL
LIN {X 0,Y 457.952,Z 738.835,A -85,B 0,C 180,E1 8457.261,E2 8457.261} C_VEL
LIN {X 0,Y 440.218,Z 887.972,A -85,B 0,C 180,E1 8455.377,E2 8455.377} C_VEL
LIN {X 0,Y 435.622,Z 914.798,A -85,B 0,C 180,E1 8455.015,E2 8455.015} C_VEL
LIN {X 0,Y 429.153,Z 941.64,A -85,B 0,C 180,E1 8454.568,E2 8454.568} C_VEL
LIN {X 0,Y 422.853,Z 962.918,A -85,B 0,C 180,E1 8454.126,E2 8454.126} C_VEL
LIN {X 0,Y 415.739,Z 983.377,A -85,B 0,C 180,E1 8453.614,E2 8453.614} C_VEL
LIN {X 0,Y 407.22,Z 1004.615,A -85,B 0,C 180,E1 8452.975,E2 8452.975} C_VEL
LIN {X 0,Y 395.301,Z 1030.264,A -85,B 0,C 180,E1 8452.037,E2 8452.037} C_VEL
LIN {X 0,Y 383.554,Z 1052.047,A -85,B 0,C 180,E1 8451.055,E2 8451.055} C_VEL
LIN {X 0,Y 372.477,Z 1070.505,A -85,B 0,C 180,E1 8450.065,E2 8450.065} C_VEL
LIN {X 0,Y 360.61,Z 1088.466,A -85,B 0,C 180,E1 8448.925,E2 8448.925} C_VEL
LIN {X 0,Y 346.199,Z 1108.298,A -85,B 0,C 180,E1 8447.427,E2 8447.427} C_VEL
LIN {X 0,Y 329.407,Z 1128.93,A -85,B 0,C 180,E1 8445.49,E2 8445.49} C_VEL
LIN {X 0,Y 315.579,Z 1144.43,A -85,B 0,C 180,E1 8443.705,E2 8443.705} C_VEL
LIN {X 0,Y 301.25,Z 1159.301,A -85,B 0,C 180,E1 8441.634,E2 8441.634} C_VEL
LIN {X 0,Y 286.53,Z 1173.485,A -85,B 0,C 180,E1 8439.23,E2 8439.23} C_VEL
LIN {X 0,Y 268.507,Z 1189.588,A -85,B 0,C 180,E1 8435.801,E2 8435.801} C_VEL
LIN {X 0,Y 252.222,Z 1202.9,A -85,B 0,C 180,E1 8432.105,E2 8432.105} C_VEL
LIN {X 0,Y 238.38,Z 1213.606,A -85,B 0,C 180,E1 8428.347,E2 8428.347} C_VEL
LIN {X 0,Y 225.612,Z 1223.046,A -85,B 0,C 180,E1 8424.173,E2 8424.173} C_VEL
LIN {X 0,Y 211.391,Z 1233.274,A -85,B 0,C 180,E1 8418.339,E2 8418.339} C_VEL
LIN {X 0,Y 198.728,Z 1242.033,A -85,B 0,C 180,E1 8411.437,E2 8411.437} C_VEL
LIN {X 0,Y 190.432,Z 1247.922,A -85,B 0,C 180,E1 8405.261,E2 8405.261} C_VEL
LIN {X 0,Y 184.248,Z 1252.567,A -85,B 0,C 180,E1 8398.863,E2 8398.863} C_VEL
LIN {X 0,Y 179.965,Z 1256.176,A -85,B 0,C 180,E1 8392.181,E2 8392.181} C_VEL
LIN {X 0,Y 177.33,Z 1258.894,A -85,B 0,C 180,E1 8385.017,E2 8385.017} C_VEL
LIN {X 0,Y 176.242,Z 1260.62,A -85,B 0,C 180,E1 8377.482,E2 8377.482} C_VEL
LIN {X 0,Y 176.038,Z 1261.149,A -85,B 0,C 180,E1 8371.287,E2 8371.287} C_VEL
LIN {X 0,Y 176.112,Z 1260.924,A -85,B 0,C 180,E1 8365.1,E2 8365.1} C_VEL
LIN {X 0,Y 176.6,Z 1259.88,A -85,B 0,C 180,E1 8358.556,E2 8358.556} C_VEL
LIN {X 0,Y 178.63,Z 1257.543,A -85,B 0,C 180,E1 8350.701,E2 8350.701} C_VEL
LIN {X 0,Y 183.494,Z 1253.228,A -85,B 0,C 180,E1 8342.04,E2 8342.04} C_VEL
LIN {X 0,Y 189.724,Z 1248.493,A -85,B 0,C 180,E1 8335.292,E2 8335.292} C_VEL
LIN {X 0,Y 197.585,Z 1242.888,A -85,B 0,C 180,E1 8329.232,E2 8329.232} C_VEL
LIN {X 0,Y 207.706,Z 1235.827,A -85,B 0,C 180,E1 8323.357,E2 8323.357} C_VEL
LIN {X 0,Y 221.967,Z 1225.868,A -85,B 0,C 180,E1 8317.109,E2 8317.109} C_VEL
LIN {X 0,Y 236.991,Z 1214.76,A -85,B 0,C 180,E1 8311.985,E2 8311.985} C_VEL
LIN {X 0,Y 250.736,Z 1204.187,A -85,B 0,C 180,E1 8308.184,E2 8308.184} C_VEL
LIN {X 0,Y 264.656,Z 1192.885,A -85,B 0,C 180,E1 8304.926,E2 8304.926} C_VEL
LIN {X 0,Y 281.691,Z 1178.175,A -85,B 0,C 180,E1 8301.55,E2 8301.55} C_VEL
LIN {X 0,Y 299.551,Z 1161.201,A -85,B 0,C 180,E1 8298.545,E2 8298.545} C_VEL
LIN {X 0,Y 313.845,Z 1146.508,A -85,B 0,C 180,E1 8296.452,E2 8296.452} C_VEL
LIN {X 0,Y 327.643,Z 1131.202,A -85,B 0,C 180,E1 8294.65,E2 8294.65} C_VEL
LIN {X 0,Y 341.32,Z 1114.755,A -85,B 0,C 180,E1 8293.036,E2 8293.036} C_VEL
LIN {X 0,Y 357.792,Z 1092.925,A -85,B 0,C 180,E1 8291.281,E2 8291.281} C_VEL
LIN {X 0,Y 371.102,Z 1073.071,A -85,B 0,C 180,E1 8289.983,E2 8289.983} C_VEL
LIN {X 0,Y 382.637,Z 1054.065,A -85,B 0,C 180,E1 8288.947,E2 8288.947} C_VEL
LIN {X 0,Y 392.879,Z 1035.35,A -85,B 0,C 180,E1 8288.079,E2 8288.079} C_VEL
LIN {X 0,Y 403.584,Z 1013.447,A -85,B 0,C 180,E1 8287.229,E2 8287.229} C_VEL
LIN {X 0,Y 414.558,Z 987.24,A -85,B 0,C 180,E1 8286.398,E2 8286.398} C_VEL
LIN {X 0,Y 422.186,Z 965.767,A -85,B 0,C 180,E1 8285.845,E2 8285.845} C_VEL
LIN {X 0,Y 428.649,Z 944.38,A -85,B 0,C 180,E1 8285.389,E2 8285.389} C_VEL
LIN {X 0,Y 434.051,Z 922.851,A -85,B 0,C 180,E1 8285.014,E2 8285.014} C_VEL
LIN {X 0,Y 439.405,Z 895.684,A -85,B 0,C 180,E1 8284.63,E2 8284.63} C_VEL
LIN {X 0,Y 444.964,Z 851.65,A -85,B 0,C 180,E1 8284.064,E2 8284.064} C_VEL
LIN {X 0,Y 458.218,Z 738.83,A -85,B 0,C 180,E1 8282.627,E2 8282.627} C_VEL
LIN {X 0,Y 458.076,Z 736.659,A -85,B 0,C 180,E1 8280.25,E2 8280.25} C_VEL
LIN {X 0,Y 458.05,Z 737.392,A -85,B 0,C 180,E1 8279.25,E2 8279.25} C_VEL
LIN {X 0,Y 458.23,Z 739.107,A -85,B 0,C 180,E1 8277.655,E2 8277.655} C_VEL
LIN {X 0,Y 456.477,Z 753.93,A -85,B 0,C 180,E1 8277.469,E2 8277.469} C_VEL
LIN {X 0,Y 455.521,Z 761.632,A -85,B 0,C 180,E1 8277.494,E2 8277.494} C_VEL
LIN {X 0,Y 452.802,Z 782.277,A -85,B 0,C 180,E1 8278.032,E2 8278.032} C_VEL
LIN {X 0,Y 451.985,Z 788.887,A -85,B 0,C 180,E1 8278.046,E2 8278.046} C_VEL
LIN {X 0,Y 439.681,Z 890.56,A -85,B 0,C 180,E1 8276.78,E2 8276.78} C_VEL
LIN {X 0,Y 434.824,Z 918.285,A -85,B 0,C 180,E1 8276.413,E2 8276.413} C_VEL
LIN {X 0,Y 428.268,Z 944.882,A -85,B 0,C 180,E1 8276.036,E2 8276.036} C_VEL
LIN {X 0,Y 421.925,Z 965.967,A -85,B 0,C 180,E1 8275.675,E2 8275.675} C_VEL
LIN {X 0,Y 414.897,Z 985.949,A -85,B 0,C 180,E1 8275.256,E2 8275.256} C_VEL
LIN {X 0,Y 406.207,Z 1007.416,A -85,B 0,C 180,E1 8274.71,E2 8274.71} C_VEL
LIN {X 0,Y 394.004,Z 1033.466,A -85,B 0,C 180,E1 8273.881,E2 8273.881} C_VEL
LIN {X 0,Y 382.309,Z 1055.041,A -85,B 0,C 180,E1 8273.027,E2 8273.027} C_VEL
LIN {X 0,Y 370.977,Z 1073.845,A -85,B 0,C 180,E1 8272.131,E2 8272.131} C_VEL
LIN {X 0,Y 359.009,Z 1091.896,A -85,B 0,C 180,E1 8271.1,E2 8271.1} C_VEL
LIN {X 0,Y 345.833,Z 1110.03,A -85,B 0,C 180,E1 8269.866,E2 8269.866} C_VEL
LIN {X 0,Y 328.143,Z 1132.045,A -85,B 0,C 180,E1 8268.016,E2 8268.016} C_VEL
LIN {X 0,Y 312.11,Z 1149.974,A -85,B 0,C 180,E1 8266.118,E2 8266.118} C_VEL
LIN {X 0,Y 297.331,Z 1165.249,A -85,B 0,C 180,E1 8264.129,E2 8264.129} C_VEL
LIN {X 0,Y 282.121,Z 1179.863,A -85,B 0,C 180,E1 8261.795,E2 8261.795} C_VEL
LIN {X 0,Y 262.655,Z 1197.146,A -85,B 0,C 180,E1 8258.278,E2 8258.278} C_VEL
LIN {X 0,Y 246.536,Z 1210.328,A -85,B 0,C 180,E1 8254.765,E2 8254.765} C_VEL
LIN {X 0,Y 232.128,Z 1221.498,A -85,B 0,C 180,E1 8250.993,E2 8250.993} C_VEL
LIN {X 0,Y 218.16,Z 1231.872,A -85,B 0,C 180,E1 8246.545,E2 8246.545} C_VEL
LIN {X 0,Y 202.809,Z 1242.958,A -85,B 0,C 180,E1 8240.29,E2 8240.29} C_VEL
LIN {X 0,Y 190.427,Z 1251.696,A -85,B 0,C 180,E1 8233.476,E2 8233.476} C_VEL
LIN {X 0,Y 182.059,Z 1257.836,A -85,B 0,C 180,E1 8227.182,E2 8227.182} C_VEL
LIN {X 0,Y 175.704,Z 1262.875,A -85,B 0,C 180,E1 8220.445,E2 8220.445} C_VEL
LIN {X 0,Y 171.202,Z 1267.008,A -85,B 0,C 180,E1 8213.051,E2 8213.051} C_VEL
LIN {X 0,Y 168.798,Z 1269.992,A -85,B 0,C 180,E1 8205.475,E2 8205.475} C_VEL
LIN {X 0,Y 168.044,Z 1271.832,A -85,B 0,C 180,E1 8197.881,E2 8197.881} C_VEL
LIN {X 0,Y 168.04,Z 1272.42,A -85,B 0,C 180,E1 8191.72,E2 8191.72} C_VEL
LIN {X 0,Y 168.031,Z 1272.248,A -85,B 0,C 180,E1 8185.921,E2 8185.921} C_VEL
LIN {X 0,Y 168.096,Z 1271.464,A -85,B 0,C 180,E1 8180.429,E2 8180.429} C_VEL
LIN {X 0,Y 168.932,Z 1269.743,A -85,B 0,C 180,E1 8173.865,E2 8173.865} C_VEL
LIN {X 0,Y 171.34,Z 1266.829,A -85,B 0,C 180,E1 8166.638,E2 8166.638} C_VEL
LIN {X 0,Y 175.679,Z 1262.861,A -85,B 0,C 180,E1 8159.585,E2 8159.585} C_VEL
LIN {X 0,Y 182.132,Z 1257.738,A -85,B 0,C 180,E1 8152.754,E2 8152.754} C_VEL
LIN {X 0,Y 191.284,Z 1251.042,A -85,B 0,C 180,E1 8145.977,E2 8145.977} C_VEL
LIN {X 0,Y 206.099,Z 1240.494,A -85,B 0,C 180,E1 8138.217,E2 8138.217} C_VEL
LIN {X 0,Y 219.364,Z 1230.891,A -85,B 0,C 180,E1 8133.025,E2 8133.025} C_VEL
LIN {X 0,Y 232.754,Z 1220.927,A -85,B 0,C 180,E1 8128.822,E2 8128.822} C_VEL
LIN {X 0,Y 247.955,Z 1209.102,A -85,B 0,C 180,E1 8124.894,E2 8124.894} C_VEL
LIN {X 0,Y 267.349,Z 1192.96,A -85,B 0,C 180,E1 8120.808,E2 8120.808} C_VEL
LIN {X 0,Y 282.869,Z 1178.987,A -85,B 0,C 180,E1 8118.076,E2 8118.076} C_VEL
LIN {X 0,Y 297.964,Z 1164.422,A -85,B 0,C 180,E1 8115.772,E2 8115.772} C_VEL
LIN {X 0,Y 313.341,Z 1148.446,A -85,B 0,C 180,E1 8113.718,E2 8113.718} C_VEL
LIN {X 0,Y 331.655,Z 1127.615,A -85,B 0,C 180,E1 8111.584,E2 8111.584} C_VEL
LIN {X 0,Y 346.703,Z 1108.561,A -85,B 0,C 180,E1 8110.037,E2 8110.037} C_VEL
LIN {X 0,Y 359.194,Z 1091.288,A -85,B 0,C 180,E1 8108.874,E2 8108.874} C_VEL
LIN {X 0,Y 371.352,Z 1072.871,A -85,B 0,C 180,E1 8107.828,E2 8107.828} C_VEL
LIN {X 0,Y 384.29,Z 1051.213,A -85,B 0,C 180,E1 8106.815,E2 8106.815} C_VEL
LIN {X 0,Y 397.431,Z 1025.979,A -85,B 0,C 180,E1 8105.867,E2 8105.867} C_VEL
LIN {X 0,Y 406.92,Z 1005.147,A -85,B 0,C 180,E1 8105.233,E2 8105.233} C_VEL
LIN {X 0,Y 414.802,Z 985.523,A -85,B 0,C 180,E1 8104.739,E2 8104.739} C_VEL
LIN {X 0,Y 422.074,Z 964.725,A -85,B 0,C 180,E1 8104.305,E2 8104.305} C_VEL
LIN {X 0,Y 428.916,Z 941.646,A -85,B 0,C 180,E1 8103.919,E2 8103.919} C_VEL
LIN {X 0,Y 435.758,Z 912.013,A -85,B 0,C 180,E1 8103.505,E2 8103.505} C_VEL
LIN {X 0,Y 439.689,Z 888.603,A -85,B 0,C 180,E1 8103.197,E2 8103.197} C_VEL
LIN {X 0,Y 456.847,Z 745.898,A -85,B 0,C 180,E1 8101.411,E2 8101.411} C_VEL
LIN {X 0,Y 456.821,Z 744.574,A -85,B 0,C 180,E1 8100,E2 8100} C_VEL
LIN {X 0,Y 456.816,Z 744.897,A -85,B 0,C 180,E1 8098.997,E2 8098.997} C_VEL
LIN {X 0,Y 456.813,Z 745.999,A -85,B 0,C 180,E1 8098.178,E2 8098.178} C_VEL
LIN {X 0,Y 439.645,Z 888.256,A -85,B 0,C 180,E1 8096.417,E2 8096.417} C_VEL
LIN {X 0,Y 434.999,Z 915.078,A -85,B 0,C 180,E1 8096.066,E2 8096.066} C_VEL
LIN {X 0,Y 428.468,Z 941.914,A -85,B 0,C 180,E1 8095.635,E2 8095.635} C_VEL
LIN {X 0,Y 422.107,Z 963.191,A -85,B 0,C 180,E1 8095.211,E2 8095.211} C_VEL
LIN {X 0,Y 414.921,Z 983.649,A -85,B 0,C 180,E1 8094.718,E2 8094.718} C_VEL
LIN {X 0,Y 406.525,Z 1004.387,A -85,B 0,C 180,E1 8094.12,E2 8094.12} C_VEL
LIN {X 0,Y 394.64,Z 1029.823,A -85,B 0,C 180,E1 8093.229,E2 8093.229} C_VEL
LIN {X 0,Y 382.376,Z 1052.319,A -85,B 0,C 180,E1 8092.257,E2 8092.257} C_VEL
LIN {X 0,Y 371.161,Z 1070.777,A -85,B 0,C 180,E1 8091.301,E2 8091.301} C_VEL
LIN {X 0,Y 359.131,Z 1088.738,A -85,B 0,C 180,E1 8090.203,E2 8090.203} C_VEL
LIN {X 0,Y 344.056,Z 1109.173,A -85,B 0,C 180,E1 8088.709,E2 8088.709} C_VEL
LIN {X 0,Y 326.797,Z 1129.932,A -85,B 0,C 180,E1 8086.808,E2 8086.808} C_VEL
LIN {X 0,Y 312.496,Z 1145.617,A -85,B 0,C 180,E1 8085.039,E2 8085.039} C_VEL
LIN {X 0,Y 297.981,Z 1160.328,A -85,B 0,C 180,E1 8083.026,E2 8083.026} C_VEL
LIN {X 0,Y 281.236,Z 1176.034,A -85,B 0,C 180,E1 8080.381,E2 8080.381} C_VEL
LIN {X 0,Y 262.079,Z 1192.355,A -85,B 0,C 180,E1 8076.815,E2 8076.815} C_VEL
LIN {X 0,Y 246.959,Z 1204.299,A -85,B 0,C 180,E1 8073.451,E2 8073.451} C_VEL
LIN {X 0,Y 232.733,Z 1214.887,A -85,B 0,C 180,E1 8069.69,E2 8069.69} C_VEL
LIN {X 0,Y 216.473,Z 1226.449,A -85,B 0,C 180,E1 8064.359,E2 8064.359} C_VEL
LIN {X 0,Y 201.602,Z 1236.331,A -85,B 0,C 180,E1 8058.046,E2 8058.046} C_VEL
LIN {X 0,Y 191.408,Z 1243.064,A -85,B 0,C 180,E1 8052.346,E2 8052.346} C_VEL
LIN {X 0,Y 183.005,Z 1248.684,A -85,B 0,C 180,E1 8046.143,E2 8046.143} C_VEL
LIN {X 0,Y 176.279,Z 1253.432,A -85,B 0,C 180,E1 8039.178,E2 8039.178} C_VEL
LIN {X 0,Y 170.961,Z 1257.772,A -85,B 0,C 180,E1 8030.169,E2 8030.169} C_VEL
LIN {X 0,Y 168.691,Z 1260.122,A -85,B 0,C 180,E1 8021.957,E2 8021.957} C_VEL
LIN {X 0,Y 168.123,Z 1261.18,A -85,B 0,C 180,E1 8015.102,E2 8015.102} C_VEL
LIN {X 0,Y 168.031,Z 1261.441,A -85,B 0,C 180,E1 8008.962,E2 8008.962} C_VEL
LIN {X 0,Y 168.246,Z 1260.971,A -85,B 0,C 180,E1 8002.472,E2 8002.472} C_VEL
LIN {X 0,Y 169.391,Z 1259.307,A -85,B 0,C 180,E1 7994.581,E2 7994.581} C_VEL
LIN {X 0,Y 172.195,Z 1256.651,A -85,B 0,C 180,E1 7987.089,E2 7987.089} C_VEL
LIN {X 0,Y 176.759,Z 1253.103,A -85,B 0,C 180,E1 7980.13,E2 7980.13} C_VEL
LIN {X 0,Y 183.317,Z 1248.52,A -85,B 0,C 180,E1 7973.505,E2 7973.505} C_VEL
LIN {X 0,Y 191.821,Z 1242.854,A -85,B 0,C 180,E1 7967.306,E2 7967.306} C_VEL
LIN {X 0,Y 203.142,Z 1235.415,A -85,B 0,C 180,E1 7961.126,E2 7961.126} C_VEL
LIN {X 0,Y 219.505,Z 1224.351,A -85,B 0,C 180,E1 7954.447,E2 7954.447} C_VEL
LIN {X 0,Y 233.368,Z 1214.529,A -85,B 0,C 180,E1 7950.045,E2 7950.045} C_VEL
LIN {X 0,Y 247.646,Z 1203.897,A -85,B 0,C 180,E1 7946.302,E2 7946.302} C_VEL
LIN {X 0,Y 262.815,Z 1191.91,A -85,B 0,C 180,E1 7942.954,E2 7942.954} C_VEL
LIN {X 0,Y 282.842,Z 1174.731,A -85,B 0,C 180,E1 7939.267,E2 7939.267} C_VEL
LIN {X 0,Y 297.875,Z 1160.637,A -85,B 0,C 180,E1 7936.909,E2 7936.909} C_VEL
LIN {X 0,Y 312.478,Z 1145.862,A -85,B 0,C 180,E1 7934.884,E2 7934.884} C_VEL
LIN {X 0,Y 327.149,Z 1129.787,A -85,B 0,C 180,E1 7933.072,E2 7933.072} C_VEL
LIN {X 0,Y 343.847,Z 1109.762,A -85,B 0,C 180,E1 7931.235,E2 7931.235} C_VEL
LIN {X 0,Y 359.139,Z 1089.079,A -85,B 0,C 180,E1 7929.718,E2 7929.718} C_VEL
LIN {X 0,Y 370.709,Z 1071.877,A -85,B 0,C 180,E1 7928.66,E2 7928.66} C_VEL
LIN {X 0,Y 381.974,Z 1053.441,A -85,B 0,C 180,E1 7927.698,E2 7927.698} C_VEL
LIN {X 0,Y 392.77,Z 1033.822,A -85,B 0,C 180,E1 7926.834,E2 7926.834} C_VEL
LIN {X 0,Y 405.129,Z 1008.278,A -85,B 0,C 180,E1 7925.909,E2 7925.909} C_VEL
LIN {X 0,Y 414.696,Z 984.941,A -85,B 0,C 180,E1 7925.221,E2 7925.221} C_VEL
LIN {X 0,Y 422.086,Z 964.055,A -85,B 0,C 180,E1 7924.715,E2 7924.715} C_VEL
LIN {X 0,Y 428.477,Z 942.82,A -85,B 0,C 180,E1 7924.287,E2 7924.287} C_VEL
LIN {X 0,Y 434.595,Z 918.082,A -85,B 0,C 180,E1 7923.883,E2 7923.883} C_VEL
LIN {X 0,Y 439.71,Z 889.697,A -85,B 0,C 180,E1 7923.509,E2 7923.509} C_VEL
LIN {X 0,Y 449.114,Z 812.702,A -85,B 0,C 180,E1 7922.55,E2 7922.55} C_VEL
LIN {X 0,Y 457.093,Z 745.963,A -85,B 0,C 180,E1 7921.724,E2 7921.724} C_VEL
LIN {X 0,Y 457.101,Z 744.599,A -85,B 0,C 180,E1 7920.251,E2 7920.251} C_VEL
LIN {X 0,Y 457.104,Z 746.093,A -85,B 0,C 180,E1 7918.574,E2 7918.574} C_VEL
LIN {X 0,Y 451.985,Z 788.887,A -85,B 0,C 180,E1 7918.046,E2 7918.046} C_VEL
LIN {X 0,Y 451.029,Z 796.591,A -85,B 0,C 180,E1 7918.077,E2 7918.077} C_VEL
LIN {X 0,Y 448.354,Z 817.23,A -85,B 0,C 180,E1 7918.626,E2 7918.626} C_VEL
LIN {X 0,Y 447.539,Z 823.839,A -85,B 0,C 180,E1 7918.642,E2 7918.642} C_VEL
LIN {X 0,Y 439.116,Z 891.63,A -85,B 0,C 180,E1 7917.813,E2 7917.813} C_VEL
LIN {X 0,Y 433.688,Z 921.039,A -85,B 0,C 180,E1 7917.434,E2 7917.434} C_VEL
LIN {X 0,Y 427.609,Z 945.26,A -85,B 0,C 180,E1 7917.103,E2 7917.103} C_VEL
LIN {X 0,Y 421.148,Z 966.454,A -85,B 0,C 180,E1 7916.756,E2 7916.756} C_VEL
LIN {X 0,Y 413.477,Z 987.884,A -85,B 0,C 180,E1 7916.323,E2 7916.323} C_VEL
LIN {X 0,Y 403.113,Z 1012.815,A -85,B 0,C 180,E1 7915.699,E2 7915.699} C_VEL
LIN {X 0,Y 391.175,Z 1037.041,A -85,B 0,C 180,E1 7914.927,E2 7914.927} C_VEL
LIN {X 0,Y 380.488,Z 1056.336,A -85,B 0,C 180,E1 7914.181,E2 7914.181} C_VEL
LIN {X 0,Y 368.873,Z 1075.246,A -85,B 0,C 180,E1 7913.306,E2 7913.306} C_VEL
LIN {X 0,Y 355.284,Z 1095.268,A -85,B 0,C 180,E1 7912.187,E2 7912.187} C_VEL
LIN {X 0,Y 337.558,Z 1118.525,A -85,B 0,C 180,E1 7910.562,E2 7910.562} C_VEL
LIN {X 0,Y 323.661,Z 1134.985,A -85,B 0,C 180,E1 7909.138,E2 7909.138} C_VEL
LIN {X 0,Y 309.13,Z 1150.838,A -85,B 0,C 180,E1 7907.484,E2 7907.484} C_VEL
LIN {X 0,Y 294.277,Z 1165.834,A -85,B 0,C 180,E1 7905.573,E2 7905.573} C_VEL
LIN {X 0,Y 276.223,Z 1182.721,A -85,B 0,C 180,E1 7902.892,E2 7902.892} C_VEL
LIN {X 0,Y 257.044,Z 1198.96,A -85,B 0,C 180,E1 7899.507,E2 7899.507} C_VEL
LIN {X 0,Y 241.522,Z 1211.223,A -85,B 0,C 180,E1 7896.215,E2 7896.215} C_VEL
LIN {X 0,Y 226.712,Z 1222.276,A -85,B 0,C 180,E1 7892.454,E2 7892.454} C_VEL
LIN {X 0,Y 209.713,Z 1234.413,A -85,B 0,C 180,E1 7887.068,E2 7887.068} C_VEL
LIN {X 0,Y 194.507,Z 1244.625,A -85,B 0,C 180,E1 7880.78,E2 7880.78} C_VEL
LIN {X 0,Y 183.469,Z 1252.048,A -85,B 0,C 180,E1 7874.688,E2 7874.688} C_VEL
LIN {X 0,Y 174.704,Z 1258.09,A -85,B 0,C 180,E1 7868.195,E2 7868.195} C_VEL
LIN {X 0,Y 167.493,Z 1263.466,A -85,B 0,C 180,E1 7860.509,E2 7860.509} C_VEL
LIN {X 0,Y 162.152,Z 1268.272,A -85,B 0,C 180,E1 7850.594,E2 7850.594} C_VEL
LIN {X 0,Y 160.313,Z 1270.763,A -85,B 0,C 180,E1 7842.259,E2 7842.259} C_VEL
LIN {X 0,Y 160.032,Z 1271.91,A -85,B 0,C 180,E1 7835.394,E2 7835.394} C_VEL
LIN {X 0,Y 160.027,Z 1272.226,A -85,B 0,C 180,E1 7829.3,E2 7829.3} C_VEL
LIN {X 0,Y 160.044,Z 1271.804,A -85,B 0,C 180,E1 7823.2,E2 7823.2} C_VEL
LIN {X 0,Y 160.719,Z 1270.077,A -85,B 0,C 180,E1 7814.871,E2 7814.871} C_VEL
LIN {X 0,Y 163.441,Z 1266.894,A -85,B 0,C 180,E1 7806.205,E2 7806.205} C_VEL
LIN {X 0,Y 168.27,Z 1262.803,A -85,B 0,C 180,E1 7798.493,E2 7798.493} C_VEL
LIN {X 0,Y 175.072,Z 1257.784,A -85,B 0,C 180,E1 7791.485,E2 7791.485} C_VEL
LIN {X 0,Y 184.094,Z 1251.573,A -85,B 0,C 180,E1 7784.917,E2 7784.917} C_VEL
LIN {X 0,Y 196.892,Z 1243.012,A -85,B 0,C 180,E1 7778.106,E2 7778.106} C_VEL
LIN {X 0,Y 213.246,Z 1231.765,A -85,B 0,C 180,E1 7771.679,E2 7771.679} C_VEL
LIN {X 0,Y 227.356,Z 1221.702,A -85,B 0,C 180,E1 7767.361,E2 7767.361} C_VEL
LIN {X 0,Y 241.445,Z 1211.165,A -85,B 0,C 180,E1 7763.797,E2 7763.797} C_VEL
LIN {X 0,Y 257.145,Z 1198.741,A -85,B 0,C 180,E1 7760.466,E2 7760.466} C_VEL
LIN {X 0,Y 276.729,Z 1182.073,A -85,B 0,C 180,E1 7757.018,E2 7757.018} C_VEL
LIN {X 0,Y 294.188,Z 1165.723,A -85,B 0,C 180,E1 7754.431,E2 7754.431} C_VEL
LIN {X 0,Y 309.228,Z 1150.514,A -85,B 0,C 180,E1 7752.495,E2 7752.495} C_VEL
LIN {X 0,Y 324.143,Z 1134.196,A -85,B 0,C 180,E1 7750.801,E2 7750.801} C_VEL
LIN {X 0,Y 341.641,Z 1113.203,A -85,B 0,C 180,E1 7749.04,E2 7749.04} C_VEL
LIN {X 0,Y 356.602,Z 1093.034,A -85,B 0,C 180,E1 7747.691,E2 7747.691} C_VEL
LIN {X 0,Y 369.372,Z 1074.078,A -85,B 0,C 180,E1 7746.643,E2 7746.643} C_VEL
LIN {X 0,Y 380.829,Z 1055.326,A -85,B 0,C 180,E1 7745.784,E2 7745.784} C_VEL
LIN {X 0,Y 393.337,Z 1032.513,A -85,B 0,C 180,E1 7744.919,E2 7744.919} C_VEL
LIN {X 0,Y 404.96,Z 1007.914,A -85,B 0,C 180,E1 7744.173,E2 7744.173} C_VEL
LIN {X 0,Y 413.724,Z 986.539,A -85,B 0,C 180,E1 7743.652,E2 7743.652} C_VEL
LIN {X 0,Y 421.055,Z 965.936,A -85,B 0,C 180,E1 7743.237,E2 7743.237} C_VEL
LIN {X 0,Y 427.581,Z 944.416,A -85,B 0,C 180,E1 7742.888,E2 7742.888} C_VEL
LIN {X 0,Y 434.27,Z 917.396,A -85,B 0,C 180,E1 7742.52,E2 7742.52} C_VEL
LIN {X 0,Y 439.085,Z 889.928,A -85,B 0,C 180,E1 7742.168,E2 7742.168} C_VEL
LIN {X 0,Y 454.798,Z 761.427,A -85,B 0,C 180,E1 7740.605,E2 7740.605} C_VEL
LIN {X 0,Y 455.832,Z 752.89,A -85,B 0,C 180,E1 7740.471,E2 7740.471} C_VEL
LIN {X 0,Y 455.854,Z 752.496,A -85,B 0,C 180,E1 7739.372,E2 7739.372} C_VEL
LIN {X 0,Y 455.806,Z 753.043,A -85,B 0,C 180,E1 7739.101,E2 7739.101} C_VEL
LIN {X 0,Y 439.202,Z 888.647,A -85,B 0,C 180,E1 7737.458,E2 7737.458} C_VEL
LIN {X 0,Y 434.432,Z 915.828,A -85,B 0,C 180,E1 7737.113,E2 7737.113} C_VEL
LIN {X 0,Y 427.872,Z 942.405,A -85,B 0,C 180,E1 7736.702,E2 7736.702} C_VEL
LIN {X 0,Y 421.512,Z 963.464,A -85,B 0,C 180,E1 7736.298,E2 7736.298} C_VEL
LIN {X 0,Y 414.319,Z 983.76,A -85,B 0,C 180,E1 7735.83,E2 7735.83} C_VEL
LIN {X 0,Y 405.778,Z 1004.659,A -85,B 0,C 180,E1 7735.252,E2 7735.252} C_VEL
LIN {X 0,Y 393.769,Z 1030.094,A -85,B 0,C 180,E1 7734.397,E2 7734.397} C_VEL
LIN {X 0,Y 381.368,Z 1052.59,A -85,B 0,C 180,E1 7733.465,E2 7733.465} C_VEL
LIN {X 0,Y 370.019,Z 1071.048,A -85,B 0,C 180,E1 7732.546,E2 7732.546} C_VEL
LIN {X 0,Y 358.489,Z 1088.079,A -85,B 0,C 180,E1 7731.551,E2 7731.551} C_VEL
LIN {X 0,Y 344.844,Z 1106.436,A -85,B 0,C 180,E1 7730.283,E2 7730.283} C_VEL
LIN {X 0,Y 326.581,Z 1128.476,A -85,B 0,C 180,E1 7728.391,E2 7728.391} C_VEL
LIN {X 0,Y 311.359,Z 1144.977,A -85,B 0,C 180,E1 7726.616,E2 7726.616} C_VEL
LIN {X 0,Y 297.327,Z 1159.016,A -85,B 0,C 180,E1 7724.785,E2 7724.785} C_VEL
LIN {X 0,Y 282.764,Z 1172.518,A -85,B 0,C 180,E1 7722.657,E2 7722.657} C_VEL
LIN {X 0,Y 266.985,Z 1186.098,A -85,B 0,C 180,E1 7720.017,E2 7720.017} C_VEL
LIN {X 0,Y 247.173,Z 1201.766,A -85,B 0,C 180,E1 7716.064,E2 7716.064} C_VEL
LIN {X 0,Y 230.994,Z 1213.513,A -85,B 0,C 180,E1 7712.128,E2 7712.128} C_VEL
LIN {X 0,Y 217.019,Z 1223.092,A -85,B 0,C 180,E1 7708.005,E2 7708.005} C_VEL
LIN {X 0,Y 203.02,Z 1232.25,A -85,B 0,C 180,E1 7702.901,E2 7702.901} C_VEL
LIN {X 0,Y 187.252,Z 1242.168,A -85,B 0,C 180,E1 7695.228,E2 7695.228} C_VEL
LIN {X 0,Y 177.537,Z 1248.224,A -85,B 0,C 180,E1 7688.672,E2 7688.672} C_VEL
LIN {X 0,Y 170.281,Z 1252.912,A -85,B 0,C 180,E1 7681.883,E2 7681.883} C_VEL
LIN {X 0,Y 165.086,Z 1256.564,A -85,B 0,C 180,E1 7674.684,E2 7674.684} C_VEL
LIN {X 0,Y 161.883,Z 1259.214,A -85,B 0,C 180,E1 7667.228,E2 7667.228} C_VEL
LIN {X 0,Y 160.492,Z 1260.766,A -85,B 0,C 180,E1 7660.392,E2 7660.392} C_VEL
LIN {X 0,Y 160.104,Z 1261.504,A -85,B 0,C 180,E1 7654.281,E2 7654.281} C_VEL
LIN {X 0,Y 160.056,Z 1261.659,A -85,B 0,C 180,E1 7648.194,E2 7648.194} C_VEL
LIN {X 0,Y 160.315,Z 1261.107,A -85,B 0,C 180,E1 7641.375,E2 7641.375} C_VEL
LIN {X 0,Y 161.665,Z 1259.466,A -85,B 0,C 180,E1 7633.455,E2 7633.455} C_VEL
LIN {X 0,Y 164.86,Z 1256.768,A -85,B 0,C 180,E1 7625.627,E2 7625.627} C_VEL
LIN {X 0,Y 169.943,Z 1253.175,A -85,B 0,C 180,E1 7618.407,E2 7618.407} C_VEL
LIN {X 0,Y 177.098,Z 1248.547,A -85,B 0,C 180,E1 7611.591,E2 7611.591} C_VEL
LIN {X 0,Y 186.234,Z 1242.848,A -85,B 0,C 180,E1 7605.288,E2 7605.288} C_VEL
LIN {X 0,Y 200.048,Z 1234.318,A -85,B 0,C 180,E1 7598.288,E2 7598.288} C_VEL
LIN {X 0,Y 215.553,Z 1224.176,A -85,B 0,C 180,E1 7592.391,E2 7592.391} C_VEL
LIN {X 0,Y 230.026,Z 1214.297,A -85,B 0,C 180,E1 7588.048,E2 7588.048} C_VEL
LIN {X 0,Y 244.942,Z 1203.525,A -85,B 0,C 180,E1 7584.349,E2 7584.349} C_VEL
LIN {X 0,Y 262.909,Z 1189.688,A -85,B 0,C 180,E1 7580.659,E2 7580.659} C_VEL
LIN {X 0,Y 281.056,Z 1174.243,A -85,B 0,C 180,E1 7577.533,E2 7577.533} C_VEL
LIN {X 0,Y 295.577,Z 1160.905,A -85,B 0,C 180,E1 7575.376,E2 7575.376} C_VEL
LIN {X 0,Y 310.464,Z 1146.13,A -85,B 0,C 180,E1 7573.414,E2 7573.414} C_VEL
LIN {X 0,Y 324.844,Z 1130.656,A -85,B 0,C 180,E1 7571.721,E2 7571.721} C_VEL
LIN {X 0,Y 341.882,Z 1110.628,A -85,B 0,C 180,E1 7569.936,E2 7569.936} C_VEL
LIN {X 0,Y 357.851,Z 1089.343,A -85,B 0,C 180,E1 7568.429,E2 7568.429} C_VEL
LIN {X 0,Y 369.594,Z 1072.106,A -85,B 0,C 180,E1 7567.411,E2 7567.411} C_VEL
LIN {X 0,Y 381.106,Z 1053.475,A -85,B 0,C 180,E1 7566.478,E2 7566.478} C_VEL
LIN {X 0,Y 392.368,Z 1033.187,A -85,B 0,C 180,E1 7565.624,E2 7565.624} C_VEL
LIN {X 0,Y 405.341,Z 1006.289,A -85,B 0,C 180,E1 7564.702,E2 7564.702} C_VEL
LIN {X 0,Y 414.041,Z 985.197,A -85,B 0,C 180,E1 7564.112,E2 7564.112} C_VEL
LIN {X 0,Y 421.46,Z 964.436,A -85,B 0,C 180,E1 7563.629,E2 7563.629} C_VEL
LIN {X 0,Y 427.868,Z 943.372,A -85,B 0,C 180,E1 7563.221,E2 7563.221} C_VEL
LIN {X 0,Y 433.82,Z 919.631,A -85,B 0,C 180,E1 7562.847,E2 7562.847} C_VEL
LIN {X 0,Y 439.212,Z 890.505,A -85,B 0,C 180,E1 7562.473,E2 7562.473} C_VEL
LIN {X 0,Y 447.606,Z 823.091,A -85,B 0,C 180,E1 7561.651,E2 7561.651} C_VEL
LIN {X 0,Y 456.092,Z 753.004,A -85,B 0,C 180,E1 7560.788,E2 7560.788} C_VEL
LIN {X 0,Y 456.122,Z 752.596,A -85,B 0,C 180,E1 7560,E2 7560} C_VEL
LIN {X 0,Y 456.063,Z 753.343,A -85,B 0,C 180,E1 7559.493,E2 7559.493} C_VEL
LIN {X 0,Y 447.539,Z 823.839,A -85,B 0,C 180,E1 7558.642,E2 7558.642} C_VEL
LIN {X 0,Y 446.586,Z 831.543,A -85,B 0,C 180,E1 7558.676,E2 7558.676} C_VEL
LIN {X 0,Y 443.956,Z 852.177,A -85,B 0,C 180,E1 7559.236,E2 7559.236} C_VEL
LIN {X 0,Y 443.142,Z 858.785,A -85,B 0,C 180,E1 7559.254,E2 7559.254} C_VEL
LIN {X 0,Y 437.821,Z 898.416,A -85,B 0,C 180,E1 7558.778,E2 7558.778} C_VEL
LIN {X 0,Y 432.444,Z 924.838,A -85,B 0,C 180,E1 7558.445,E2 7558.445} C_VEL
LIN {X 0,Y 426.757,Z 946.838,A -85,B 0,C 180,E1 7558.156,E2 7558.156} C_VEL
LIN {X 0,Y 420.074,Z 968.292,A -85,B 0,C 180,E1 7557.817,E2 7557.817} C_VEL
LIN {X 0,Y 410.433,Z 994.407,A -85,B 0,C 180,E1 7557.297,E2 7557.297} C_VEL
LIN {X 0,Y 399.648,Z 1018.626,A -85,B 0,C 180,E1 7556.681,E2 7556.681} C_VEL
LIN {X 0,Y 389.406,Z 1038.887,A -85,B 0,C 180,E1 7556.047,E2 7556.047} C_VEL
LIN {X 0,Y 378.131,Z 1058.802,A -85,B 0,C 180,E1 7555.298,E2 7555.298} C_VEL
LIN {X 0,Y 364.29,Z 1080.722,A -85,B 0,C 180,E1 7554.293,E2 7554.293} C_VEL
LIN {X 0,Y 348.081,Z 1103.291,A -85,B 0,C 180,E1 7553,E2 7553} C_VEL
LIN {X 0,Y 333.931,Z 1121.089,A -85,B 0,C 180,E1 7551.736,E2 7551.736} C_VEL
LIN {X 0,Y 320.194,Z 1136.939,A -85,B 0,C 180,E1 7550.383,E2 7550.383} C_VEL
LIN {X 0,Y 304.898,Z 1153.184,A -85,B 0,C 180,E1 7548.708,E2 7548.708} C_VEL
LIN {X 0,Y 285.175,Z 1172.312,A -85,B 0,C 180,E1 7546.206,E2 7546.206} C_VEL
LIN {X 0,Y 267.854,Z 1187.502,A -85,B 0,C 180,E1 7543.635,E2 7543.635} C_VEL
LIN {X 0,Y 251.931,Z 1200.479,A -85,B 0,C 180,E1 7540.861,E2 7540.861} C_VEL
LIN {X 0,Y 235.887,Z 1212.704,A -85,B 0,C 180,E1 7537.549,E2 7537.549} C_VEL
LIN {X 0,Y 217.088,Z 1226.142,A -85,B 0,C 180,E1 7532.761,E2 7532.761} C_VEL
LIN {X 0,Y 200.608,Z 1237.061,A -85,B 0,C 180,E1 7527.408,E2 7527.408} C_VEL
LIN {X 0,Y 187.734,Z 1245.322,A -85,B 0,C 180,E1 7522.042,E2 7522.042} C_VEL
LIN {X 0,Y 176.599,Z 1252.401,A -85,B 0,C 180,E1 7515.995,E2 7515.995} C_VEL
LIN {X 0,Y 165.891,Z 1259.403,A -85,B 0,C 180,E1 7507.954,E2 7507.954} C_VEL
LIN {X 0,Y 157.65,Z 1265.223,A -85,B 0,C 180,E1 7498.163,E2 7498.163} C_VEL
LIN {X 0,Y 153.936,Z 1268.488,A -85,B 0,C 180,E1 7490.154,E2 7490.154} C_VEL
LIN {X 0,Y 152.337,Z 1270.57,A -85,B 0,C 180,E1 7482.526,E2 7482.526} C_VEL
LIN {X 0,Y 152.038,Z 1271.646,A -85,B 0,C 180,E1 7475.678,E2 7475.678} C_VEL
LIN {X 0,Y 152.033,Z 1271.986,A -85,B 0,C 180,E1 7469.64,E2 7469.64} C_VEL
LIN {X 0,Y 152.047,Z 1271.566,A -85,B 0,C 180,E1 7463.22,E2 7463.22} C_VEL
LIN {X 0,Y 152.777,Z 1269.929,A -85,B 0,C 180,E1 7454.454,E2 7454.454} C_VEL
LIN {X 0,Y 155.908,Z 1266.621,A -85,B 0,C 180,E1 7444.978,E2 7444.978} C_VEL
LIN {X 0,Y 161.351,Z 1262.431,A -85,B 0,C 180,E1 7436.782,E2 7436.782} C_VEL
LIN {X 0,Y 168.962,Z 1257.265,A -85,B 0,C 180,E1 7429.409,E2 7429.409} C_VEL
LIN {X 0,Y 179.089,Z 1250.767,A -85,B 0,C 180,E1 7422.499,E2 7422.499} C_VEL
LIN {X 0,Y 194.233,Z 1241.186,A -85,B 0,C 180,E1 7415.092,E2 7415.092} C_VEL
LIN {X 0,Y 209.949,Z 1230.789,A -85,B 0,C 180,E1 7409.376,E2 7409.376} C_VEL
LIN {X 0,Y 224.342,Z 1220.896,A -85,B 0,C 180,E1 7405.243,E2 7405.243} C_VEL
LIN {X 0,Y 239.745,Z 1209.715,A -85,B 0,C 180,E1 7401.595,E2 7401.595} C_VEL
LIN {X 0,Y 259.326,Z 1194.542,A -85,B 0,C 180,E1 7397.8,E2 7397.8} C_VEL
LIN {X 0,Y 278.121,Z 1178.432,A -85,B 0,C 180,E1 7394.788,E2 7394.788} C_VEL
LIN {X 0,Y 293.108,Z 1164.588,A -85,B 0,C 180,E1 7392.728,E2 7392.728} C_VEL
LIN {X 0,Y 308.441,Z 1149.299,A -85,B 0,C 180,E1 7390.874,E2 7390.874} C_VEL
LIN {X 0,Y 325.469,Z 1130.842,A -85,B 0,C 180,E1 7389.069,E2 7389.069} C_VEL
LIN {X 0,Y 343.261,Z 1109.239,A -85,B 0,C 180,E1 7387.407,E2 7387.407} C_VEL
LIN {X 0,Y 356.595,Z 1091.345,A -85,B 0,C 180,E1 7386.297,E2 7386.297} C_VEL
LIN {X 0,Y 368.994,Z 1073.064,A -85,B 0,C 180,E1 7385.34,E2 7385.34} C_VEL
LIN {X 0,Y 381.545,Z 1052.602,A -85,B 0,C 180,E1 7384.46,E2 7384.46} C_VEL
LIN {X 0,Y 395.647,Z 1026.368,A -85,B 0,C 180,E1 7383.552,E2 7383.552} C_VEL
LIN {X 0,Y 405.449,Z 1005.324,A -85,B 0,C 180,E1 7382.969,E2 7382.969} C_VEL
LIN {X 0,Y 413.78,Z 984.974,A -85,B 0,C 180,E1 7382.505,E2 7382.505} C_VEL
LIN {X 0,Y 421.169,Z 964.177,A -85,B 0,C 180,E1 7382.114,E2 7382.114} C_VEL
LIN {X 0,Y 428.255,Z 940.61,A -85,B 0,C 180,E1 7381.761,E2 7381.761} C_VEL
LIN {X 0,Y 435.101,Z 911.289,A -85,B 0,C 180,E1 7381.384,E2 7381.384} C_VEL
LIN {X 0,Y 439.085,Z 888.031,A -85,B 0,C 180,E1 7381.097,E2 7381.097} C_VEL
LIN {X 0,Y 452.537,Z 779.431,A -85,B 0,C 180,E1 7379.801,E2 7379.801} C_VEL
LIN {X 0,Y 438.874,Z 889.252,A -85,B 0,C 180,E1 7378.499,E2 7378.499} C_VEL
LIN {X 0,Y 433.945,Z 916.819,A -85,B 0,C 180,E1 7378.16,E2 7378.16} C_VEL
LIN {X 0,Y 427.424,Z 942.895,A -85,B 0,C 180,E1 7377.772,E2 7377.772} C_VEL
LIN {X 0,Y 421.07,Z 963.737,A -85,B 0,C 180,E1 7377.388,E2 7377.388} C_VEL
LIN {X 0,Y 413.757,Z 984.176,A -85,B 0,C 180,E1 7376.937,E2 7376.937} C_VEL
LIN {X 0,Y 405.19,Z 1004.931,A -85,B 0,C 180,E1 7376.388,E2 7376.388} C_VEL
LIN {X 0,Y 393.062,Z 1030.365,A -85,B 0,C 180,E1 7375.57,E2 7375.57} C_VEL
LIN {X 0,Y 380.53,Z 1052.862,A -85,B 0,C 180,E1 7374.679,E2 7374.679} C_VEL
LIN {X 0,Y 368.751,Z 1071.782,A -85,B 0,C 180,E1 7373.773,E2 7373.773} C_VEL
LIN {X 0,Y 356.717,Z 1089.282,A -85,B 0,C 180,E1 7372.788,E2 7372.788} C_VEL
LIN {X 0,Y 341.2,Z 1109.753,A -85,B 0,C 180,E1 7371.405,E2 7371.405} C_VEL
LIN {X 0,Y 323.805,Z 1130.081,A -85,B 0,C 180,E1 7369.683,E2 7369.683} C_VEL
LIN {X 0,Y 308.654,Z 1146.164,A -85,B 0,C 180,E1 7367.995,E2 7367.995} C_VEL
LIN {X 0,Y 294.382,Z 1160.122,A -85,B 0,C 180,E1 7366.217,E2 7366.217} C_VEL
LIN {X 0,Y 278.684,Z 1174.309,A -85,B 0,C 180,E1 7364.015,E2 7364.015} C_VEL
LIN {X 0,Y 259.287,Z 1190.412,A -85,B 0,C 180,E1 7360.832,E2 7360.832} C_VEL
LIN {X 0,Y 241.544,Z 1203.726,A -85,B 0,C 180,E1 7357.351,E2 7357.351} C_VEL
LIN {X 0,Y 226.266,Z 1214.431,A -85,B 0,C 180,E1 7353.743,E2 7353.743} C_VEL
LIN {X 0,Y 211.937,Z 1223.872,A -85,B 0,C 180,E1 7349.667,E2 7349.667} C_VEL
LIN {X 0,Y 195.633,Z 1234.1,A -85,B 0,C 180,E1 7343.83,E2 7343.83} C_VEL
LIN {X 0,Y 180.772,Z 1242.846,A -85,B 0,C 180,E1 7336.695,E2 7336.695} C_VEL
LIN {X 0,Y 170.716,Z 1248.741,A -85,B 0,C 180,E1 7330.088,E2 7330.088} C_VEL
LIN {X 0,Y 163.007,Z 1253.381,A -85,B 0,C 180,E1 7323.067,E2 7323.067} C_VEL
LIN {X 0,Y 157.235,Z 1257.138,A -85,B 0,C 180,E1 7315.198,E2 7315.198} C_VEL
LIN {X 0,Y 153.676,Z 1259.911,A -85,B 0,C 180,E1 7306.617,E2 7306.617} C_VEL
LIN {X 0,Y 152.251,Z 1261.613,A -85,B 0,C 180,E1 7297.397,E2 7297.397} C_VEL
LIN {X 0,Y 152.043,Z 1262.003,A -85,B 0,C 180,E1 7290.36,E2 7290.36} C_VEL
LIN {X 0,Y 152.188,Z 1261.674,A -85,B 0,C 180,E1 7283.57,E2 7283.57} C_VEL
LIN {X 0,Y 153.289,Z 1260.362,A -85,B 0,C 180,E1 7274.859,E2 7274.859} C_VEL
LIN {X 0,Y 157.002,Z 1257.341,A -85,B 0,C 180,E1 7265.128,E2 7265.128} C_VEL
LIN {X 0,Y 162.652,Z 1253.643,A -85,B 0,C 180,E1 7257.233,E2 7257.233} C_VEL
LIN {X 0,Y 170.255,Z 1249.064,A -85,B 0,C 180,E1 7250.18,E2 7250.18} C_VEL
LIN {X 0,Y 179.9,Z 1243.413,A -85,B 0,C 180,E1 7243.718,E2 7243.718} C_VEL
LIN {X 0,Y 192.582,Z 1235.96,A -85,B 0,C 180,E1 7237.385,E2 7237.385} C_VEL
LIN {X 0,Y 210.514,Z 1224.896,A -85,B 0,C 180,E1 7230.698,E2 7230.698} C_VEL
LIN {X 0,Y 225.873,Z 1214.809,A -85,B 0,C 180,E1 7226.275,E2 7226.275} C_VEL
LIN {X 0,Y 240.887,Z 1204.324,A -85,B 0,C 180,E1 7222.708,E2 7222.708} C_VEL
LIN {X 0,Y 257.611,Z 1191.828,A -85,B 0,C 180,E1 7219.387,E2 7219.387} C_VEL
LIN {X 0,Y 277.811,Z 1175.271,A -85,B 0,C 180,E1 7216.037,E2 7216.037} C_VEL
LIN {X 0,Y 293.775,Z 1160.909,A -85,B 0,C 180,E1 7213.783,E2 7213.783} C_VEL
LIN {X 0,Y 308.657,Z 1146.397,A -85,B 0,C 180,E1 7211.926,E2 7211.926} C_VEL
LIN {X 0,Y 323.765,Z 1130.387,A -85,B 0,C 180,E1 7210.243,E2 7210.243} C_VEL
LIN {X 0,Y 341.248,Z 1110.015,A -85,B 0,C 180,E1 7208.513,E2 7208.513} C_VEL
LIN {X 0,Y 356.745,Z 1089.607,A -85,B 0,C 180,E1 7207.131,E2 7207.131} C_VEL
LIN {X 0,Y 368.612,Z 1072.401,A -85,B 0,C 180,E1 7206.16,E2 7206.16} C_VEL
LIN {X 0,Y 379.98,Z 1054.231,A -85,B 0,C 180,E1 7205.284,E2 7205.284} C_VEL
LIN {X 0,Y 391.174,Z 1034.342,A -85,B 0,C 180,E1 7204.48,E2 7204.48} C_VEL
LIN {X 0,Y 403.787,Z 1008.793,A -85,B 0,C 180,E1 7203.63,E2 7203.63} C_VEL
LIN {X 0,Y 413.542,Z 985.453,A -85,B 0,C 180,E1 7203,E2 7203} C_VEL
LIN {X 0,Y 421.135,Z 964.369,A -85,B 0,C 180,E1 7202.532,E2 7202.532} C_VEL
LIN {X 0,Y 427.639,Z 943.109,A -85,B 0,C 180,E1 7202.139,E2 7202.139} C_VEL
LIN {X 0,Y 434.082,Z 917.412,A -85,B 0,C 180,E1 7201.756,E2 7201.756} C_VEL
LIN {X 0,Y 439.089,Z 889.708,A -85,B 0,C 180,E1 7201.416,E2 7201.416} C_VEL
LIN {X 0,Y 450.482,Z 798.515,A -85,B 0,C 180,E1 7200.332,E2 7200.332} C_VEL
LIN {X 0,Y 452.334,Z 783.425,A -85,B 0,C 180,E1 7200.148,E2 7200.148} C_VEL
LIN {X 0,Y 443.142,Z 858.785,A -85,B 0,C 180,E1 7199.254,E2 7199.254} C_VEL
LIN {X 0,Y 442.211,Z 866.485,A -85,B 0,C 180,E1 7199.294,E2 7199.294} C_VEL
LIN {X 0,Y 439.401,Z 887.084,A -85,B 0,C 180,E1 7199.867,E2 7199.867} C_VEL
LIN {X 0,Y 438.428,Z 893.675,A -85,B 0,C 180,E1 7199.885,E2 7199.885} C_VEL
LIN {X 0,Y 432.736,Z 922.758,A -85,B 0,C 180,E1 7199.534,E2 7199.534} C_VEL
LIN {X 0,Y 426.897,Z 945.455,A -85,B 0,C 180,E1 7199.252,E2 7199.252} C_VEL
LIN {X 0,Y 420.408,Z 966.349,A -85,B 0,C 180,E1 7198.947,E2 7198.947} C_VEL
LIN {X 0,Y 412.606,Z 987.756,A -85,B 0,C 180,E1 7198.558,E2 7198.558} C_VEL
LIN {X 0,Y 401.728,Z 1013.314,A -85,B 0,C 180,E1 7197.98,E2 7197.98} C_VEL
LIN {X 0,Y 389.911,Z 1036.812,A -85,B 0,C 180,E1 7197.304,E2 7197.304} C_VEL
LIN {X 0,Y 379.134,Z 1055.885,A -85,B 0,C 180,E1 7196.637,E2 7196.637} C_VEL
LIN {X 0,Y 367.366,Z 1074.65,A -85,B 0,C 180,E1 7195.853,E2 7195.853} C_VEL
LIN {X 0,Y 353.904,Z 1094.063,A -85,B 0,C 180,E1 7194.869,E2 7194.869} C_VEL
LIN {X 0,Y 336.193,Z 1116.867,A -85,B 0,C 180,E1 7193.435,E2 7193.435} C_VEL
LIN {X 0,Y 320.613,Z 1134.805,A -85,B 0,C 180,E1 7192.025,E2 7192.025} C_VEL
LIN {X 0,Y 305.577,Z 1150.673,A -85,B 0,C 180,E1 7190.495,E2 7190.495} C_VEL
LIN {X 0,Y 289.585,Z 1166.214,A -85,B 0,C 180,E1 7188.649,E2 7188.649} C_VEL
LIN {X 0,Y 269.995,Z 1183.666,A -85,B 0,C 180,E1 7186.023,E2 7186.023} C_VEL
LIN {X 0,Y 250.986,Z 1198.91,A -85,B 0,C 180,E1 7182.989,E2 7182.989} C_VEL
LIN {X 0,Y 235.221,Z 1210.672,A -85,B 0,C 180,E1 7179.981,E2 7179.981} C_VEL
LIN {X 0,Y 219.297,Z 1221.799,A -85,B 0,C 180,E1 7176.344,E2 7176.344} C_VEL
LIN {X 0,Y 201.01,Z 1233.86,A -85,B 0,C 180,E1 7171.123,E2 7171.123} C_VEL
LIN {X 0,Y 184.503,Z 1243.953,A -85,B 0,C 180,E1 7164.937,E2 7164.937} C_VEL
LIN {X 0,Y 171.898,Z 1251.497,A -85,B 0,C 180,E1 7158.641,E2 7158.641} C_VEL
LIN {X 0,Y 161.428,Z 1257.806,A -85,B 0,C 180,E1 7151.529,E2 7151.529} C_VEL
LIN {X 0,Y 151.89,Z 1263.994,A -85,B 0,C 180,E1 7141.797,E2 7141.797} C_VEL
LIN {X 0,Y 146.392,Z 1268.097,A -85,B 0,C 180,E1 7131.661,E2 7131.661} C_VEL
LIN {X 0,Y 144.411,Z 1270.303,A -85,B 0,C 180,E1 7123.226,E2 7123.226} C_VEL
LIN {X 0,Y 144.042,Z 1271.383,A -85,B 0,C 180,E1 7115.995,E2 7115.995} C_VEL
LIN {X 0,Y 144.037,Z 1271.724,A -85,B 0,C 180,E1 7109.62,E2 7109.62} C_VEL
LIN {X 0,Y 144.055,Z 1271.302,A -85,B 0,C 180,E1 7102.842,E2 7102.842} C_VEL
LIN {X 0,Y 144.922,Z 1269.661,A -85,B 0,C 180,E1 7093.588,E2 7093.588} C_VEL
LIN {X 0,Y 148.465,Z 1266.339,A -85,B 0,C 180,E1 7083.603,E2 7083.603} C_VEL
LIN {X 0,Y 154.284,Z 1262.254,A -85,B 0,C 180,E1 7075.251,E2 7075.251} C_VEL
LIN {X 0,Y 162.677,Z 1256.989,A -85,B 0,C 180,E1 7067.484,E2 7067.484} C_VEL
LIN {X 0,Y 173.444,Z 1250.524,A -85,B 0,C 180,E1 7060.478,E2 7060.478} C_VEL
LIN {X 0,Y 189.495,Z 1240.907,A -85,B 0,C 180,E1 7052.998,E2 7052.998} C_VEL
LIN {X 0,Y 205.914,Z 1230.525,A -85,B 0,C 180,E1 7047.333,E2 7047.333} C_VEL
LIN {X 0,Y 220.871,Z 1220.617,A -85,B 0,C 180,E1 7043.26,E2 7043.26} C_VEL
LIN {X 0,Y 236.77,Z 1209.437,A -85,B 0,C 180,E1 7039.697,E2 7039.697} C_VEL
LIN {X 0,Y 256.576,Z 1194.514,A -85,B 0,C 180,E1 7036.063,E2 7036.063} C_VEL
LIN {X 0,Y 275.211,Z 1178.937,A -85,B 0,C 180,E1 7033.228,E2 7033.228} C_VEL
LIN {X 0,Y 290.472,Z 1165.168,A -85,B 0,C 180,E1 7031.234,E2 7031.234} C_VEL
LIN {X 0,Y 306.052,Z 1149.961,A -85,B 0,C 180,E1 7029.445,E2 7029.445} C_VEL
LIN {X 0,Y 321.721,Z 1133.338,A -85,B 0,C 180,E1 7027.86,E2 7027.86} C_VEL
LIN {X 0,Y 339.909,Z 1112.037,A -85,B 0,C 180,E1 7026.237,E2 7026.237} C_VEL
LIN {X 0,Y 355.256,Z 1091.812,A -85,B 0,C 180,E1 7025.018,E2 7025.018} C_VEL
LIN {X 0,Y 367.835,Z 1073.53,A -85,B 0,C 180,E1 7024.103,E2 7024.103} C_VEL
LIN {X 0,Y 379.598,Z 1054.665,A -85,B 0,C 180,E1 7023.322,E2 7023.322} C_VEL
LIN {X 0,Y 392.767,Z 1031.062,A -85,B 0,C 180,E1 7022.519,E2 7022.519} C_VEL
LIN {X 0,Y 404.788,Z 1005.791,A -85,B 0,C 180,E1 7021.84,E2 7021.84} C_VEL
LIN {X 0,Y 413.479,Z 984.768,A -85,B 0,C 180,E1 7021.386,E2 7021.386} C_VEL
LIN {X 0,Y 420.949,Z 963.903,A -85,B 0,C 180,E1 7021.016,E2 7021.016} C_VEL
LIN {X 0,Y 428.073,Z 940.37,A -85,B 0,C 180,E1 7020.684,E2 7020.684} C_VEL
LIN {X 0,Y 434.95,Z 911.171,A -85,B 0,C 180,E1 7020.325,E2 7020.325} C_VEL
LIN {X 0,Y 438.989,Z 887.852,A -85,B 0,C 180,E1 7020.047,E2 7020.047} C_VEL
LIN {X 0,Y 441.747,Z 867.306,A -85,B 0,C 180,E1 7019.804,E2 7019.804} C_VEL
LIN {X 0,Y 436.623,Z 902.318,A -85,B 0,C 180,E1 7019.394,E2 7019.394} C_VEL
LIN {X 0,Y 431.777,Z 925.394,A -85,B 0,C 180,E1 7019.108,E2 7019.108} C_VEL
LIN {X 0,Y 426.182,Z 946.674,A -85,B 0,C 180,E1 7018.79,E2 7018.79} C_VEL
LIN {X 0,Y 419.298,Z 968.427,A -85,B 0,C 180,E1 7018.395,E2 7018.395} C_VEL
LIN {X 0,Y 409.188,Z 995.087,A -85,B 0,C 180,E1 7017.794,E2 7017.794} C_VEL
LIN {X 0,Y 398.966,Z 1017.665,A -85,B 0,C 180,E1 7017.164,E2 7017.164} C_VEL
LIN {X 0,Y 389.103,Z 1036.891,A -85,B 0,C 180,E1 7016.527,E2 7016.527} C_VEL
LIN {X 0,Y 378.519,Z 1055.366,A -85,B 0,C 180,E1 7015.802,E2 7015.802} C_VEL
LIN {X 0,Y 366.337,Z 1074.505,A -85,B 0,C 180,E1 7014.911,E2 7014.911} C_VEL
LIN {X 0,Y 350.709,Z 1096.532,A -85,B 0,C 180,E1 7013.67,E2 7013.67} C_VEL
LIN {X 0,Y 334.552,Z 1116.562,A -85,B 0,C 180,E1 7012.271,E2 7012.271} C_VEL
LIN {X 0,Y 320.433,Z 1132.509,A -85,B 0,C 180,E1 7010.919,E2 7010.919} C_VEL
LIN {X 0,Y 306.131,Z 1147.351,A -85,B 0,C 180,E1 7009.396,E2 7009.396} C_VEL
LIN {X 0,Y 290.728,Z 1162.062,A -85,B 0,C 180,E1 7007.564,E2 7007.564} C_VEL
LIN {X 0,Y 271.275,Z 1179.073,A -85,B 0,C 180,E1 7004.901,E2 7004.901} C_VEL
LIN {X 0,Y 252.462,Z 1193.803,A -85,B 0,C 180,E1 7001.86,E2 7001.86} C_VEL
LIN {X 0,Y 236.848,Z 1205.124,A -85,B 0,C 180,E1 6998.865,E2 6998.865} C_VEL
LIN {X 0,Y 221.938,Z 1215.21,A -85,B 0,C 180,E1 6995.479,E2 6995.479} C_VEL
LIN {X 0,Y 206.42,Z 1225.042,A -85,B 0,C 180,E1 6991.221,E2 6991.221} C_VEL
LIN {X 0,Y 187.666,Z 1236.128,A -85,B 0,C 180,E1 6984.577,E2 6984.577} C_VEL
LIN {X 0,Y 174.291,Z 1243.594,A -85,B 0,C 180,E1 6978.201,E2 6978.201} C_VEL
LIN {X 0,Y 164.008,Z 1249.259,A -85,B 0,C 180,E1 6971.622,E2 6971.622} C_VEL
LIN {X 0,Y 155.469,Z 1254.048,A -85,B 0,C 180,E1 6964.001,E2 6964.001} C_VEL
LIN {X 0,Y 148.571,Z 1258.318,A -85,B 0,C 180,E1 6954.218,E2 6954.218} C_VEL
LIN {X 0,Y 145.036,Z 1260.919,A -85,B 0,C 180,E1 6943.943,E2 6943.943} C_VEL
LIN {X 0,Y 144.169,Z 1261.97,A -85,B 0,C 180,E1 6935.953,E2 6935.953} C_VEL
LIN {X 0,Y 144.042,Z 1262.251,A -85,B 0,C 180,E1 6929.186,E2 6929.186} C_VEL
LIN {X 0,Y 144.287,Z 1261.878,A -85,B 0,C 180,E1 6922.015,E2 6922.015} C_VEL
LIN {X 0,Y 145.889,Z 1260.214,A -85,B 0,C 180,E1 6912.431,E2 6912.431} C_VEL
LIN {X 0,Y 149.819,Z 1257.458,A -85,B 0,C 180,E1 6903.421,E2 6903.421} C_VEL
LIN {X 0,Y 156.119,Z 1253.716,A -85,B 0,C 180,E1 6895.231,E2 6895.231} C_VEL
LIN {X 0,Y 164.704,Z 1248.935,A -85,B 0,C 180,E1 6887.786,E2 6887.786} C_VEL
LIN {X 0,Y 176.435,Z 1242.514,A -85,B 0,C 180,E1 6880.57,E2 6880.57} C_VEL
LIN {X 0,Y 193.376,Z 1232.918,A -85,B 0,C 180,E1 6873.087,E2 6873.087} C_VEL
LIN {X 0,Y 208.527,Z 1223.826,A -85,B 0,C 180,E1 6868.061,E2 6868.061} C_VEL
LIN {X 0,Y 223.735,Z 1214.145,A -85,B 0,C 180,E1 6863.997,E2 6863.997} C_VEL
LIN {X 0,Y 240.872,Z 1202.466,A -85,B 0,C 180,E1 6860.234,E2 6860.234} C_VEL
LIN {X 0,Y 261.76,Z 1186.83,A -85,B 0,C 180,E1 6856.483,E2 6856.483} C_VEL
LIN {X 0,Y 278.268,Z 1173.266,A -85,B 0,C 180,E1 6854.002,E2 6854.002} C_VEL
LIN {X 0,Y 293.694,Z 1159.532,A -85,B 0,C 180,E1 6851.986,E2 6851.986} C_VEL
LIN {X 0,Y 309.816,Z 1143.923,A -85,B 0,C 180,E1 6850.123,E2 6850.123} C_VEL
LIN {X 0,Y 329.31,Z 1122.989,A -85,B 0,C 180,E1 6848.143,E2 6848.143} C_VEL
LIN {X 0,Y 344.392,Z 1104.861,A -85,B 0,C 180,E1 6846.774,E2 6846.774} C_VEL
LIN {X 0,Y 357.737,Z 1087.225,A -85,B 0,C 180,E1 6845.672,E2 6845.672} C_VEL
LIN {X 0,Y 370.241,Z 1069.02,A -85,B 0,C 180,E1 6844.724,E2 6844.724} C_VEL
LIN {X 0,Y 384.229,Z 1046.335,A -85,B 0,C 180,E1 6843.73,E2 6843.73} C_VEL
LIN {X 0,Y 396.917,Z 1022.399,A -85,B 0,C 180,E1 6842.888,E2 6842.888} C_VEL
LIN {X 0,Y 406.304,Z 1002.309,A -85,B 0,C 180,E1 6842.302,E2 6842.302} C_VEL
LIN {X 0,Y 414.728,Z 981.75,A -85,B 0,C 180,E1 6841.796,E2 6841.796} C_VEL
LIN {X 0,Y 422.86,Z 958.664,A -85,B 0,C 180,E1 6841.326,E2 6841.326} C_VEL
LIN {X 0,Y 430.866,Z 930.393,A -85,B 0,C 180,E1 6840.868,E2 6840.868} C_VEL
LIN {X 0,Y 435.9,Z 907.571,A -85,B 0,C 180,E1 6840.577,E2 6840.577} C_VEL
LIN {X 0,Y 439.634,Z 885.352,A -85,B 0,C 180,E1 6840.317,E2 6840.317} C_VEL
LIN {X 0,Y 441.554,Z 871.226,A -85,B 0,C 180,E1 6840.147,E2 6840.147} C_VEL
LIN {X 0,Y 438.428,Z 893.675,A -85,B 0,C 180,E1 6839.885,E2 6839.885} C_VEL
LIN {X 0,Y 438.404,Z 894.011,A -85,B 0,C 180,E1 6839.883,E2 6839.883} C_VEL
LIN {X 0,Y 438.404,Z 976.425,A -85,B 0,C 180,E1 6839.883,E2 6839.883} C_VEL
LIN {X 0,Y 429.295,Z 976.425,A -85,B 0,C 180,E1 6840.255,E2 6840.255} C_VEL
LIN {X 0,Y 427.386,Z 974.425,A -85,B 0,C 180,E1 6840.335,E2 6840.335} C_VEL
LIN {X 0,Y 427.386,Z 956.912,A -85,B 0,C 180,E1 6840.335,E2 6840.335} C_VEL
LIN {X 0,Y 423.654,Z 956.249,A -85,B 0,C 180,E1 6840.189,E2 6840.189} C_VEL
LIN {X 0,Y 414.978,Z 981.05,A -85,B 0,C 180,E1 6839.801,E2 6839.801} C_VEL
LIN {X 0,Y 406.499,Z 1001.837,A -85,B 0,C 180,E1 6839.392,E2 6839.392} C_VEL
LIN {X 0,Y 397.547,Z 1021.136,A -85,B 0,C 180,E1 6838.934,E2 6838.934} C_VEL
LIN {X 0,Y 387.138,Z 1041.08,A -85,B 0,C 180,E1 6838.362,E2 6838.362} C_VEL
LIN {X 0,Y 373.327,Z 1064.61,A -85,B 0,C 180,E1 6837.538,E2 6837.538} C_VEL
LIN {X 0,Y 358.282,Z 1086.863,A -85,B 0,C 180,E1 6836.553,E2 6836.553} C_VEL
LIN {X 0,Y 344.519,Z 1105.213,A -85,B 0,C 180,E1 6835.565,E2 6835.565} C_VEL
LIN {X 0,Y 330.485,Z 1122.27,A -85,B 0,C 180,E1 6834.444,E2 6834.444} C_VEL
LIN {X 0,Y 315.275,Z 1139.171,A -85,B 0,C 180,E1 6833.102,E2 6833.102} C_VEL
LIN {X 0,Y 294.613,Z 1159.876,A -85,B 0,C 180,E1 6831.013,E2 6831.013} C_VEL
LIN {X 0,Y 277.326,Z 1175.472,A -85,B 0,C 180,E1 6828.984,E2 6828.984} C_VEL
LIN {X 0,Y 261.829,Z 1188.379,A -85,B 0,C 180,E1 6826.887,E2 6826.887} C_VEL
LIN {X 0,Y 245.192,Z 1201.224,A -85,B 0,C 180,E1 6824.266,E2 6824.266} C_VEL
LIN {X 0,Y 225.029,Z 1215.652,A -85,B 0,C 180,E1 6820.415,E2 6820.415} C_VEL
LIN {X 0,Y 206.035,Z 1227.944,A -85,B 0,C 180,E1 6815.858,E2 6815.858} C_VEL
LIN {X 0,Y 190.615,Z 1237.342,A -85,B 0,C 180,E1 6811.188,E2 6811.188} C_VEL
LIN {X 0,Y 176.576,Z 1245.499,A -85,B 0,C 180,E1 6805.788,E2 6805.788} C_VEL
LIN {X 0,Y 162.108,Z 1253.734,A -85,B 0,C 180,E1 6798.294,E2 6798.294} C_VEL
LIN {X 0,Y 149.745,Z 1260.698,A -85,B 0,C 180,E1 6788.898,E2 6788.898} C_VEL
LIN {X 0,Y 142.569,Z 1265.079,A -85,B 0,C 180,E1 6780.348,E2 6780.348} C_VEL
LIN {X 0,Y 138.308,Z 1268.192,A -85,B 0,C 180,E1 6771.655,E2 6771.655} C_VEL
LIN {X 0,Y 136.446,Z 1270.111,A -85,B 0,C 180,E1 6763.581,E2 6763.581} C_VEL
LIN {X 0,Y 136.045,Z 1271.145,A -85,B 0,C 180,E1 6755.925,E2 6755.925} C_VEL
LIN {X 0,Y 136.041,Z 1271.461,A -85,B 0,C 180,E1 6749.598,E2 6749.598} C_VEL
LIN {X 0,Y 136.059,Z 1271.062,A -85,B 0,C 180,E1 6742.8,E2 6742.8} C_VEL
LIN {X 0,Y 136.919,Z 1269.583,A -85,B 0,C 180,E1 6733.474,E2 6733.474} C_VEL
LIN {X 0,Y 140.865,Z 1266.241,A -85,B 0,C 180,E1 6722.533,E2 6722.533} C_VEL
LIN {X 0,Y 147.145,Z 1262.195,A -85,B 0,C 180,E1 6713.783,E2 6713.783} C_VEL
LIN {X 0,Y 156.118,Z 1256.977,A -85,B 0,C 180,E1 6705.751,E2 6705.751} C_VEL
LIN {X 0,Y 166.954,Z 1250.874,A -85,B 0,C 180,E1 6698.899,E2 6698.899} C_VEL
LIN {X 0,Y 181.031,Z 1242.906,A -85,B 0,C 180,E1 6692.353,E2 6692.353} C_VEL
LIN {X 0,Y 200.677,Z 1231.187,A -85,B 0,C 180,E1 6685.635,E2 6685.635} C_VEL
LIN {X 0,Y 216.875,Z 1220.865,A -85,B 0,C 180,E1 6681.402,E2 6681.402} C_VEL
LIN {X 0,Y 232.636,Z 1210.153,A -85,B 0,C 180,E1 6678.027,E2 6678.027} C_VEL
LIN {X 0,Y 249.437,Z 1197.906,A -85,B 0,C 180,E1 6675.022,E2 6675.022} C_VEL
LIN {X 0,Y 270.028,Z 1181.595,A -85,B 0,C 180,E1 6671.968,E2 6671.968} C_VEL
LIN {X 0,Y 288.036,Z 1165.748,A -85,B 0,C 180,E1 6669.714,E2 6669.714} C_VEL
LIN {X 0,Y 303.856,Z 1150.622,A -85,B 0,C 180,E1 6667.994,E2 6667.994} C_VEL
LIN {X 0,Y 318.978,Z 1134.906,A -85,B 0,C 180,E1 6666.543,E2 6666.543} C_VEL
LIN {X 0,Y 334.292,Z 1117.534,A -85,B 0,C 180,E1 6665.235,E2 6665.235} C_VEL
LIN {X 0,Y 352.197,Z 1094.906,A -85,B 0,C 180,E1 6663.868,E2 6663.868} C_VEL
LIN {X 0,Y 366.358,Z 1074.738,A -85,B 0,C 180,E1 6662.89,E2 6662.89} C_VEL
LIN {X 0,Y 378.157,Z 1056.14,A -85,B 0,C 180,E1 6662.152,E2 6662.152} C_VEL
LIN {X 0,Y 389.025,Z 1037.128,A -85,B 0,C 180,E1 6661.52,E2 6661.52} C_VEL
LIN {X 0,Y 400.436,Z 1014.704,A -85,B 0,C 180,E1 6660.905,E2 6660.905} C_VEL
LIN {X 0,Y 411.891,Z 988.299,A -85,B 0,C 180,E1 6660.336,E2 6660.336} C_VEL
LIN {X 0,Y 419.883,Z 966.598,A -85,B 0,C 180,E1 6659.962,E2 6659.962} C_VEL
LIN {X 0,Y 424.2,Z 953.482,A -85,B 0,C 180,E1 6659.765,E2 6659.765} C_VEL
LIN {X 0,Y 414.919,Z 980.329,A -85,B 0,C 180,E1 6659.258,E2 6659.258} C_VEL
LIN {X 0,Y 406.477,Z 1000.978,A -85,B 0,C 180,E1 6658.782,E2 6658.782} C_VEL
LIN {X 0,Y 397.076,Z 1021.113,A -85,B 0,C 180,E1 6658.23,E2 6658.23} C_VEL
LIN {X 0,Y 386.238,Z 1041.63,A -85,B 0,C 180,E1 6657.562,E2 6657.562} C_VEL
LIN {X 0,Y 371.552,Z 1066.036,A -85,B 0,C 180,E1 6656.584,E2 6656.584} C_VEL
LIN {X 0,Y 357.455,Z 1086.52,A -85,B 0,C 180,E1 6655.584,E2 6655.584} C_VEL
LIN {X 0,Y 343.959,Z 1104.242,A -85,B 0,C 180,E1 6654.536,E2 6654.536} C_VEL
LIN {X 0,Y 330.111,Z 1120.801,A -85,B 0,C 180,E1 6653.363,E2 6653.363} C_VEL
LIN {X 0,Y 312.19,Z 1140.301,A -85,B 0,C 180,E1 6651.677,E2 6651.677} C_VEL
LIN {X 0,Y 293.637,Z 1158.172,A -85,B 0,C 180,E1 6649.701,E2 6649.701} C_VEL
LIN {X 0,Y 277.27,Z 1172.584,A -85,B 0,C 180,E1 6647.702,E2 6647.702} C_VEL
LIN {X 0,Y 261.277,Z 1185.546,A -85,B 0,C 180,E1 6645.462,E2 6645.462} C_VEL
LIN {X 0,Y 242.334,Z 1199.687,A -85,B 0,C 180,E1 6642.341,E2 6642.341} C_VEL
LIN {X 0,Y 221.778,Z 1213.473,A -85,B 0,C 180,E1 6638.201,E2 6638.201} C_VEL
LIN {X 0,Y 206.253,Z 1223.082,A -85,B 0,C 180,E1 6634.347,E2 6634.347} C_VEL
LIN {X 0,Y 191.758,Z 1231.5,A -85,B 0,C 180,E1 6629.916,E2 6629.916} C_VEL
LIN {X 0,Y 177.835,Z 1239.142,A -85,B 0,C 180,E1 6624.584,E2 6624.584} C_VEL
LIN {X 0,Y 162.371,Z 1247.333,A -85,B 0,C 180,E1 6616.579,E2 6616.579} C_VEL
LIN {X 0,Y 150.576,Z 1253.333,A -85,B 0,C 180,E1 6607.632,E2 6607.632} C_VEL
LIN {X 0,Y 143.314,Z 1257.224,A -85,B 0,C 180,E1 6599.212,E2 6599.212} C_VEL
LIN {X 0,Y 139.012,Z 1259.805,A -85,B 0,C 180,E1 6591.057,E2 6591.057} C_VEL
LIN {X 0,Y 136.847,Z 1261.437,A -85,B 0,C 180,E1 6583.071,E2 6583.071} C_VEL
LIN {X 0,Y 136.169,Z 1262.253,A -85,B 0,C 180,E1 6575.881,E2 6575.881} C_VEL
LIN {X 0,Y 136.054,Z 1262.491,A -85,B 0,C 180,E1 6568.718,E2 6568.718} C_VEL
LIN {X 0,Y 136.344,Z 1262.091,A -85,B 0,C 180,E1 6561.122,E2 6561.122} C_VEL
LIN {X 0,Y 138.148,Z 1260.481,A -85,B 0,C 180,E1 6551.411,E2 6551.411} C_VEL
LIN {X 0,Y 142.515,Z 1257.727,A -85,B 0,C 180,E1 6541.942,E2 6541.942} C_VEL
LIN {X 0,Y 149.404,Z 1253.987,A -85,B 0,C 180,E1 6533.423,E2 6533.423} C_VEL
LIN {X 0,Y 158.828,Z 1249.118,A -85,B 0,C 180,E1 6525.65,E2 6525.65} C_VEL
LIN {X 0,Y 171.724,Z 1242.494,A -85,B 0,C 180,E1 6518.161,E2 6518.161} C_VEL
LIN {X 0,Y 189.642,Z 1232.796,A -85,B 0,C 180,E1 6510.727,E2 6510.727} C_VEL
LIN {X 0,Y 204.728,Z 1224.099,A -85,B 0,C 180,E1 6505.996,E2 6505.996} C_VEL
LIN {X 0,Y 220.165,Z 1214.611,A -85,B 0,C 180,E1 6502.085,E2 6502.085} C_VEL
LIN {X 0,Y 237.282,Z 1203.299,A -85,B 0,C 180,E1 6498.51,E2 6498.51} C_VEL
LIN {X 0,Y 259.525,Z 1187.1,A -85,B 0,C 180,E1 6494.723,E2 6494.723} C_VEL
LIN {X 0,Y 276.493,Z 1173.44,A -85,B 0,C 180,E1 6492.32,E2 6492.32} C_VEL
LIN {X 0,Y 291.82,Z 1160.045,A -85,B 0,C 180,E1 6490.431,E2 6490.431} C_VEL
LIN {X 0,Y 307.542,Z 1145.104,A -85,B 0,C 180,E1 6488.712,E2 6488.712} C_VEL
LIN {X 0,Y 325.879,Z 1125.998,A -85,B 0,C 180,E1 6486.941,E2 6486.941} C_VEL
LIN {X 0,Y 342.564,Z 1106.33,A -85,B 0,C 180,E1 6485.499,E2 6485.499} C_VEL
LIN {X 0,Y 356.055,Z 1088.812,A -85,B 0,C 180,E1 6484.443,E2 6484.443} C_VEL
LIN {X 0,Y 367.997,Z 1071.767,A -85,B 0,C 180,E1 6483.583,E2 6483.583} C_VEL
LIN {X 0,Y 379.925,Z 1052.956,A -85,B 0,C 180,E1 6482.768,E2 6482.768} C_VEL
LIN {X 0,Y 393.203,Z 1029.49,A -85,B 0,C 180,E1 6481.934,E2 6481.934} C_VEL
LIN {X 0,Y 405.069,Z 1004.814,A -85,B 0,C 180,E1 6481.223,E2 6481.223} C_VEL
LIN {X 0,Y 413.51,Z 984.687,A -85,B 0,C 180,E1 6480.742,E2 6480.742} C_VEL
LIN {X 0,Y 420.981,Z 964.141,A -85,B 0,C 180,E1 6480.333,E2 6480.333} C_VEL
LIN {X 0,Y 423.654,Z 956.249,A -85,B 0,C 180,E1 6480.189,E2 6480.189} C_VEL
LIN {X 0,Y 426.894,Z 956.999,A -85,B 0,C 180,E1 6479.908,E2 6479.908} C_VEL
LIN {X 0,Y 426.894,Z 1028.435,A -85,B 0,C 180,E1 6479.908,E2 6479.908} C_VEL
LIN {X 0,Y 406.829,Z 1028.435,A -85,B 0,C 180,E1 6480.397,E2 6480.397} C_VEL
LIN {X 0,Y 404.861,Z 1026.435,A -85,B 0,C 180,E1 6480.447,E2 6480.447} C_VEL
LIN {X 0,Y 404.861,Z 1014.161,A -85,B 0,C 180,E1 6480.447,E2 6480.447} C_VEL
LIN {X 0,Y 401.263,Z 1013.238,A -85,B 0,C 180,E1 6480.286,E2 6480.286} C_VEL
LIN {X 0,Y 389.608,Z 1036.065,A -85,B 0,C 180,E1 6479.706,E2 6479.706} C_VEL
LIN {X 0,Y 378.215,Z 1055.872,A -85,B 0,C 180,E1 6479.091,E2 6479.091} C_VEL
LIN {X 0,Y 366.129,Z 1074.743,A -85,B 0,C 180,E1 6478.387,E2 6478.387} C_VEL
LIN {X 0,Y 351.847,Z 1094.854,A -85,B 0,C 180,E1 6477.467,E2 6477.467} C_VEL
LIN {X 0,Y 333.731,Z 1117.452,A -85,B 0,C 180,E1 6476.179,E2 6476.179} C_VEL
LIN {X 0,Y 318.231,Z 1134.799,A -85,B 0,C 180,E1 6474.943,E2 6474.943} C_VEL
LIN {X 0,Y 302.752,Z 1150.643,A -85,B 0,C 180,E1 6473.553,E2 6473.553} C_VEL
LIN {X 0,Y 285.898,Z 1166.462,A -85,B 0,C 180,E1 6471.832,E2 6471.832} C_VEL
LIN {X 0,Y 263.695,Z 1185.256,A -85,B 0,C 180,E1 6469.174,E2 6469.174} C_VEL
LIN {X 0,Y 245.628,Z 1199.061,A -85,B 0,C 180,E1 6466.583,E2 6466.583} C_VEL
LIN {X 0,Y 229.135,Z 1210.708,A -85,B 0,C 180,E1 6463.774,E2 6463.774} C_VEL
LIN {X 0,Y 211.559,Z 1222.226,A -85,B 0,C 180,E1 6460.168,E2 6460.168} C_VEL
LIN {X 0,Y 189.561,Z 1235.441,A -85,B 0,C 180,E1 6454.372,E2 6454.372} C_VEL
LIN {X 0,Y 173.632,Z 1244.323,A -85,B 0,C 180,E1 6448.783,E2 6448.783} C_VEL
LIN {X 0,Y 160.069,Z 1251.574,A -85,B 0,C 180,E1 6442.519,E2 6442.519} C_VEL
LIN {X 0,Y 147.351,Z 1258.316,A -85,B 0,C 180,E1 6434.363,E2 6434.363} C_VEL
LIN {X 0,Y 136.258,Z 1264.365,A -85,B 0,C 180,E1 6423.221,E2 6423.221} C_VEL
LIN {X 0,Y 130.859,Z 1267.8,A -85,B 0,C 180,E1 6413.432,E2 6413.432} C_VEL
LIN {X 0,Y 128.547,Z 1269.844,A -85,B 0,C 180,E1 6404.433,E2 6404.433} C_VEL
LIN {X 0,Y 128.052,Z 1270.881,A -85,B 0,C 180,E1 6396.296,E2 6396.296} C_VEL
LIN {X 0,Y 128.045,Z 1271.199,A -85,B 0,C 180,E1 6389.573,E2 6389.573} C_VEL
LIN {X 0,Y 128.056,Z 1270.799,A -85,B 0,C 180,E1 6382.393,E2 6382.393} C_VEL
LIN {X 0,Y 129.099,Z 1269.314,A -85,B 0,C 180,E1 6372.441,E2 6372.441} C_VEL
LIN {X 0,Y 133.564,Z 1265.974,A -85,B 0,C 180,E1 6360.907,E2 6360.907} C_VEL
LIN {X 0,Y 140.486,Z 1261.92,A -85,B 0,C 180,E1 6351.768,E2 6351.768} C_VEL
LIN {X 0,Y 150.205,Z 1256.7,A -85,B 0,C 180,E1 6343.511,E2 6343.511} C_VEL
LIN {X 0,Y 161.794,Z 1250.597,A -85,B 0,C 180,E1 6336.575,E2 6336.575} C_VEL
LIN {X 0,Y 177.483,Z 1242.187,A -85,B 0,C 180,E1 6329.721,E2 6329.721} C_VEL
LIN {X 0,Y 197.171,Z 1230.908,A -85,B 0,C 180,E1 6323.422,E2 6323.422} C_VEL
LIN {X 0,Y 213.936,Z 1220.585,A -85,B 0,C 180,E1 6319.294,E2 6319.294} C_VEL
LIN {X 0,Y 229.909,Z 1210.05,A -85,B 0,C 180,E1 6316.077,E2 6316.077} C_VEL
LIN {X 0,Y 247.39,Z 1197.627,A -85,B 0,C 180,E1 6313.14,E2 6313.14} C_VEL
LIN {X 0,Y 268.185,Z 1181.512,A -85,B 0,C 180,E1 6310.245,E2 6310.245} C_VEL
LIN {X 0,Y 287.385,Z 1164.886,A -85,B 0,C 180,E1 6308,E2 6308} C_VEL
LIN {X 0,Y 303.287,Z 1149.877,A -85,B 0,C 180,E1 6306.389,E2 6306.389} C_VEL
LIN {X 0,Y 318.24,Z 1134.522,A -85,B 0,C 180,E1 6305.047,E2 6305.047} C_VEL
LIN {X 0,Y 334.228,Z 1116.579,A -85,B 0,C 180,E1 6303.774,E2 6303.774} C_VEL
LIN {X 0,Y 352.77,Z 1093.217,A -85,B 0,C 180,E1 6302.46,E2 6302.46} C_VEL
LIN {X 0,Y 366.036,Z 1074.464,A -85,B 0,C 180,E1 6301.607,E2 6301.607} C_VEL
LIN {X 0,Y 378.005,Z 1055.756,A -85,B 0,C 180,E1 6300.909,E2 6300.909} C_VEL
LIN {X 0,Y 389.386,Z 1035.962,A -85,B 0,C 180,E1 6300.294,E2 6300.294} C_VEL
LIN {X 0,Y 401.893,Z 1011.362,A -85,B 0,C 180,E1 6299.668,E2 6299.668} C_VEL
LIN {X 0,Y 389.525,Z 1035.515,A -85,B 0,C 180,E1 6298.97,E2 6298.97} C_VEL
LIN {X 0,Y 378.555,Z 1054.48,A -85,B 0,C 180,E1 6298.312,E2 6298.312} C_VEL
LIN {X 0,Y 366.752,Z 1072.826,A -85,B 0,C 180,E1 6297.551,E2 6297.551} C_VEL
LIN {X 0,Y 353.988,Z 1090.76,A -85,B 0,C 180,E1 6296.68,E2 6296.68} C_VEL
LIN {X 0,Y 336.977,Z 1112.296,A -85,B 0,C 180,E1 6295.405,E2 6295.405} C_VEL
LIN {X 0,Y 319.194,Z 1132.07,A -85,B 0,C 180,E1 6293.923,E2 6293.923} C_VEL
LIN {X 0,Y 304.477,Z 1146.983,A -85,B 0,C 180,E1 6292.544,E2 6292.544} C_VEL
LIN {X 0,Y 289.479,Z 1160.944,A -85,B 0,C 180,E1 6290.988,E2 6290.988} C_VEL
LIN {X 0,Y 272.581,Z 1175.385,A -85,B 0,C 180,E1 6289.003,E2 6289.003} C_VEL
LIN {X 0,Y 251.316,Z 1191.86,A -85,B 0,C 180,E1 6286.059,E2 6286.059} C_VEL
LIN {X 0,Y 233.066,Z 1204.552,A -85,B 0,C 180,E1 6283.029,E2 6283.029} C_VEL
LIN {X 0,Y 216.361,Z 1215.258,A -85,B 0,C 180,E1 6279.698,E2 6279.698} C_VEL
LIN {X 0,Y 200.433,Z 1224.712,A -85,B 0,C 180,E1 6275.853,E2 6275.853} C_VEL
LIN {X 0,Y 181.989,Z 1234.926,A -85,B 0,C 180,E1 6270.202,E2 6270.202} C_VEL
LIN {X 0,Y 164.704,Z 1243.643,A -85,B 0,C 180,E1 6263.057,E2 6263.057} C_VEL
LIN {X 0,Y 152.513,Z 1249.561,A -85,B 0,C 180,E1 6256.123,E2 6256.123} C_VEL
LIN {X 0,Y 142.471,Z 1254.395,A -85,B 0,C 180,E1 6248.115,E2 6248.115} C_VEL
LIN {X 0,Y 134.527,Z 1258.403,A -85,B 0,C 180,E1 6238.38,E2 6238.38} C_VEL
LIN {X 0,Y 129.564,Z 1261.328,A -85,B 0,C 180,E1 6226.569,E2 6226.569} C_VEL
LIN {X 0,Y 128.241,Z 1262.477,A -85,B 0,C 180,E1 6217.145,E2 6217.145} C_VEL
LIN {X 0,Y 128.053,Z 1262.798,A -85,B 0,C 180,E1 6209.532,E2 6209.532} C_VEL
LIN {X 0,Y 128.305,Z 1262.44,A -85,B 0,C 180,E1 6201.78,E2 6201.78} C_VEL
LIN {X 0,Y 130.17,Z 1260.962,A -85,B 0,C 180,E1 6191.159,E2 6191.159} C_VEL
LIN {X 0,Y 135.311,Z 1257.997,A -85,B 0,C 180,E1 6180.303,E2 6180.303} C_VEL
LIN {X 0,Y 142.842,Z 1254.258,A -85,B 0,C 180,E1 6171.444,E2 6171.444} C_VEL
LIN {X 0,Y 152.995,Z 1249.39,A -85,B 0,C 180,E1 6163.474,E2 6163.474} C_VEL
LIN {X 0,Y 166.699,Z 1242.767,A -85,B 0,C 180,E1 6155.906,E2 6155.906} C_VEL
LIN {X 0,Y 185.519,Z 1233.068,A -85,B 0,C 180,E1 6148.512,E2 6148.512} C_VEL
LIN {X 0,Y 201.205,Z 1224.371,A -85,B 0,C 180,E1 6143.857,E2 6143.857} C_VEL
LIN {X 0,Y 217.164,Z 1214.883,A -85,B 0,C 180,E1 6140.044,E2 6140.044} C_VEL
LIN {X 0,Y 234.785,Z 1203.561,A -85,B 0,C 180,E1 6136.579,E2 6136.579} C_VEL
LIN {X 0,Y 257.54,Z 1187.37,A -85,B 0,C 180,E1 6132.937,E2 6132.937} C_VEL
LIN {X 0,Y 274.729,Z 1173.805,A -85,B 0,C 180,E1 6130.646,E2 6130.646} C_VEL
LIN {X 0,Y 290.437,Z 1160.313,A -85,B 0,C 180,E1 6128.827,E2 6128.827} C_VEL
LIN {X 0,Y 306.403,Z 1145.371,A -85,B 0,C 180,E1 6127.19,E2 6127.19} C_VEL
LIN {X 0,Y 324.99,Z 1126.264,A -85,B 0,C 180,E1 6125.506,E2 6125.506} C_VEL
LIN {X 0,Y 341.878,Z 1106.594,A -85,B 0,C 180,E1 6124.135,E2 6124.135} C_VEL
LIN {X 0,Y 355.517,Z 1089.075,A -85,B 0,C 180,E1 6123.132,E2 6123.132} C_VEL
LIN {X 0,Y 367.781,Z 1071.73,A -85,B 0,C 180,E1 6122.305,E2 6122.305} C_VEL
LIN {X 0,Y 379.619,Z 1053.217,A -85,B 0,C 180,E1 6121.546,E2 6121.546} C_VEL
LIN {X 0,Y 393.013,Z 1029.749,A -85,B 0,C 180,E1 6120.755,E2 6120.755} C_VEL
LIN {X 0,Y 401.263,Z 1013.238,A -85,B 0,C 180,E1 6120.286,E2 6120.286} C_VEL
LIN {X 0,Y 404.649,Z 1014.208,A -85,B 0,C 180,E1 6120.057,E2 6120.057} C_VEL
LIN {X 0,Y 404.649,Z 1068.16,A -85,B 0,C 180,E1 6120.057,E2 6120.057} C_VEL
LIN {X 0,Y 384.143,Z 1068.16,A -85,B 0,C 180,E1 6120.523,E2 6120.523} C_VEL
LIN {X 0,Y 382.169,Z 1066.16,A -85,B 0,C 180,E1 6120.571,E2 6120.571} C_VEL
LIN {X 0,Y 382.169,Z 1055.739,A -85,B 0,C 180,E1 6120.571,E2 6120.571} C_VEL
LIN {X 0,Y 378.771,Z 1054.635,A -85,B 0,C 180,E1 6120.363,E2 6120.363} C_VEL
LIN {X 0,Y 366.988,Z 1072.998,A -85,B 0,C 180,E1 6119.727,E2 6119.727} C_VEL
LIN {X 0,Y 354.044,Z 1091.245,A -85,B 0,C 180,E1 6118.963,E2 6118.963} C_VEL
LIN {X 0,Y 336.728,Z 1113.255,A -85,B 0,C 180,E1 6117.839,E2 6117.839} C_VEL
LIN {X 0,Y 318.582,Z 1133.504,A -85,B 0,C 180,E1 6116.512,E2 6116.512} C_VEL
LIN {X 0,Y 303.048,Z 1149.288,A -85,B 0,C 180,E1 6115.22,E2 6115.22} C_VEL
LIN {X 0,Y 287.689,Z 1163.619,A -85,B 0,C 180,E1 6113.782,E2 6113.782} C_VEL
LIN {X 0,Y 270.653,Z 1178.226,A -85,B 0,C 180,E1 6111.972,E2 6111.972} C_VEL
LIN {X 0,Y 248.434,Z 1195.5,A -85,B 0,C 180,E1 6109.164,E2 6109.164} C_VEL
LIN {X 0,Y 229.566,Z 1208.677,A -85,B 0,C 180,E1 6106.271,E2 6106.271} C_VEL
LIN {X 0,Y 212.224,Z 1219.844,A -85,B 0,C 180,E1 6103.056,E2 6103.056} C_VEL
LIN {X 0,Y 194.848,Z 1230.216,A -85,B 0,C 180,E1 6099.09,E2 6099.09} C_VEL
LIN {X 0,Y 174.583,Z 1241.421,A -85,B 0,C 180,E1 6093.098,E2 6093.098} C_VEL
LIN {X 0,Y 157.615,Z 1250.042,A -85,B 0,C 180,E1 6086.231,E2 6086.231} C_VEL
LIN {X 0,Y 145.133,Z 1256.186,A -85,B 0,C 180,E1 6079.298,E2 6079.298} C_VEL
LIN {X 0,Y 134.899,Z 1261.234,A -85,B 0,C 180,E1 6071.298,E2 6071.298} C_VEL
LIN {X 0,Y 127.252,Z 1265.211,A -85,B 0,C 180,E1 6062.32,E2 6062.32} C_VEL
LIN {X 0,Y 122.446,Z 1268.138,A -85,B 0,C 180,E1 6052.591,E2 6052.591} C_VEL
LIN {X 0,Y 120.305,Z 1270.021,A -85,B 0,C 180,E1 6042.501,E2 6042.501} C_VEL
LIN {X 0,Y 120.05,Z 1270.746,A -85,B 0,C 180,E1 6034.321,E2 6034.321} C_VEL
LIN {X 0,Y 120.06,Z 1270.843,A -85,B 0,C 180,E1 6027.635,E2 6027.635} C_VEL
LIN {X 0,Y 120.119,Z 1270.381,A -85,B 0,C 180,E1 6019.955,E2 6019.955} C_VEL
LIN {X 0,Y 121.814,Z 1268.609,A -85,B 0,C 180,E1 6009.35,E2 6009.35} C_VEL
LIN {X 0,Y 126.786,Z 1265.449,A -85,B 0,C 180,E1 5998.402,E2 5998.402} C_VEL
LIN {X 0,Y 134.433,Z 1261.428,A -85,B 0,C 180,E1 5989.145,E2 5989.145} C_VEL
LIN {X 0,Y 144.559,Z 1256.414,A -85,B 0,C 180,E1 5981.079,E2 5981.079} C_VEL
LIN {X 0,Y 156.915,Z 1250.319,A -85,B 0,C 180,E1 5974.102,E2 5974.102} C_VEL
LIN {X 0,Y 172.569,Z 1242.349,A -85,B 0,C 180,E1 5967.602,E2 5967.602} C_VEL
LIN {X 0,Y 193.966,Z 1230.629,A -85,B 0,C 180,E1 5961.131,E2 5961.131} C_VEL
LIN {X 0,Y 211.293,Z 1220.306,A -85,B 0,C 180,E1 5957.13,E2 5957.13} C_VEL
LIN {X 0,Y 228.288,Z 1209.392,A -85,B 0,C 180,E1 5953.94,E2 5953.94} C_VEL
LIN {X 0,Y 245.614,Z 1197.349,A -85,B 0,C 180,E1 5951.228,E2 5951.228} C_VEL
LIN {X 0,Y 266.82,Z 1181.234,A -85,B 0,C 180,E1 5948.471,E2 5948.471} C_VEL
LIN {X 0,Y 285.692,Z 1165.195,A -85,B 0,C 180,E1 5946.409,E2 5946.409} C_VEL
LIN {X 0,Y 301.991,Z 1150.069,A -85,B 0,C 180,E1 5944.864,E2 5944.864} C_VEL
LIN {X 0,Y 317.514,Z 1134.354,A -85,B 0,C 180,E1 5943.563,E2 5943.563} C_VEL
LIN {X 0,Y 333.681,Z 1116.422,A -85,B 0,C 180,E1 5942.363,E2 5942.363} C_VEL
LIN {X 0,Y 352.261,Z 1093.283,A -85,B 0,C 180,E1 5941.138,E2 5941.138} C_VEL
LIN {X 0,Y 366.085,Z 1073.913,A -85,B 0,C 180,E1 5940.313,E2 5940.313} C_VEL
LIN {X 0,Y 377.896,Z 1055.593,A -85,B 0,C 180,E1 5939.674,E2 5939.674} C_VEL
LIN {X 0,Y 379.388,Z 1053.16,A -85,B 0,C 180,E1 5939.595,E2 5939.595} C_VEL
LIN {X 0,Y 367.462,Z 1071.677,A -85,B 0,C 180,E1 5938.88,E2 5938.88} C_VEL
LIN {X 0,Y 354.517,Z 1089.815,A -85,B 0,C 180,E1 5938.06,E2 5938.06} C_VEL
LIN {X 0,Y 339.359,Z 1109.001,A -85,B 0,C 180,E1 5937.009,E2 5937.009} C_VEL
LIN {X 0,Y 319.883,Z 1130.84,A -85,B 0,C 180,E1 5935.508,E2 5935.508} C_VEL
LIN {X 0,Y 304.261,Z 1146.549,A -85,B 0,C 180,E1 5934.153,E2 5934.153} C_VEL
LIN {X 0,Y 288.518,Z 1161.026,A -85,B 0,C 180,E1 5932.633,E2 5932.633} C_VEL
LIN {X 0,Y 271.432,Z 1175.407,A -85,B 0,C 180,E1 5930.759,E2 5930.759} C_VEL
LIN {X 0,Y 250.054,Z 1191.714,A -85,B 0,C 180,E1 5927.999,E2 5927.999} C_VEL
LIN {X 0,Y 230.054,Z 1205.289,A -85,B 0,C 180,E1 5924.884,E2 5924.884} C_VEL
LIN {X 0,Y 213.609,Z 1215.533,A -85,B 0,C 180,E1 5921.797,E2 5921.797} C_VEL
LIN {X 0,Y 197.186,Z 1224.975,A -85,B 0,C 180,E1 5918.074,E2 5918.074} C_VEL
LIN {X 0,Y 177.995,Z 1235.2,A -85,B 0,C 180,E1 5912.531,E2 5912.531} C_VEL
LIN {X 0,Y 160.024,Z 1243.832,A -85,B 0,C 180,E1 5905.533,E2 5905.533} C_VEL
LIN {X 0,Y 146.877,Z 1249.835,A -85,B 0,C 180,E1 5898.459,E2 5898.459} C_VEL
LIN {X 0,Y 136.054,Z 1254.667,A -85,B 0,C 180,E1 5890.267,E2 5890.267} C_VEL
LIN {X 0,Y 127.352,Z 1258.673,A -85,B 0,C 180,E1 5880.139,E2 5880.139} C_VEL
LIN {X 0,Y 121.795,Z 1261.595,A -85,B 0,C 180,E1 5867.66,E2 5867.66} C_VEL
LIN {X 0,Y 120.272,Z 1262.741,A -85,B 0,C 180,E1 5857.622,E2 5857.622} C_VEL
LIN {X 0,Y 120.057,Z 1263.06,A -85,B 0,C 180,E1 5849.501,E2 5849.501} C_VEL
LIN {X 0,Y 120.332,Z 1262.71,A -85,B 0,C 180,E1 5841.377,E2 5841.377} C_VEL
LIN {X 0,Y 122.485,Z 1261.229,A -85,B 0,C 180,E1 5829.927,E2 5829.927} C_VEL
LIN {X 0,Y 128.228,Z 1258.266,A -85,B 0,C 180,E1 5818.481,E2 5818.481} C_VEL
LIN {X 0,Y 136.46,Z 1254.529,A -85,B 0,C 180,E1 5809.275,E2 5809.275} C_VEL
LIN {X 0,Y 147.396,Z 1249.662,A -85,B 0,C 180,E1 5801.127,E2 5801.127} C_VEL
LIN {X 0,Y 162.603,Z 1242.747,A -85,B 0,C 180,E1 5793.224,E2 5793.224} C_VEL
LIN {X 0,Y 181.678,Z 1233.341,A -85,B 0,C 180,E1 5786.196,E2 5786.196} C_VEL
LIN {X 0,Y 198.046,Z 1224.604,A -85,B 0,C 180,E1 5781.627,E2 5781.627} C_VEL
LIN {X 0,Y 214.668,Z 1215.024,A -85,B 0,C 180,E1 5777.904,E2 5777.904} C_VEL
LIN {X 0,Y 233.41,Z 1203.28,A -85,B 0,C 180,E1 5774.468,E2 5774.468} C_VEL
LIN {X 0,Y 255.81,Z 1187.64,A -85,B 0,C 180,E1 5771.125,E2 5771.125} C_VEL
LIN {X 0,Y 273.32,Z 1174.074,A -85,B 0,C 180,E1 5768.94,E2 5768.94} C_VEL
LIN {X 0,Y 289.284,Z 1160.582,A -85,B 0,C 180,E1 5767.21,E2 5767.21} C_VEL
LIN {X 0,Y 305.786,Z 1145.349,A -85,B 0,C 180,E1 5765.63,E2 5765.63} C_VEL
LIN {X 0,Y 324.792,Z 1125.981,A -85,B 0,C 180,E1 5764.025,E2 5764.025} C_VEL
LIN {X 0,Y 341.877,Z 1106.256,A -85,B 0,C 180,E1 5762.733,E2 5762.733} C_VEL
LIN {X 0,Y 355.164,Z 1089.338,A -85,B 0,C 180,E1 5761.819,E2 5761.819} C_VEL
LIN {X 0,Y 368.04,Z 1071.263,A -85,B 0,C 180,E1 5761.008,E2 5761.008} C_VEL
LIN {X 0,Y 378.771,Z 1054.635,A -85,B 0,C 180,E1 5760.363,E2 5760.363} C_VEL
LIN {X 0,Y 382.2,Z 1055.74,A -85,B 0,C 180,E1 5760.167,E2 5760.167} C_VEL
LIN {X 0,Y 382.2,Z 1100.08,A -85,B 0,C 180,E1 5760.167,E2 5760.167} C_VEL
LIN {X 0,Y 361.619,Z 1100.08,A -85,B 0,C 180,E1 5760.576,E2 5760.576} C_VEL
LIN {X 0,Y 359.636,Z 1098.08,A -85,B 0,C 180,E1 5760.618,E2 5760.618} C_VEL
LIN {X 0,Y 359.636,Z 1089.148,A -85,B 0,C 180,E1 5760.618,E2 5760.618} C_VEL
LIN {X 0,Y 356.276,Z 1087.907,A -85,B 0,C 180,E1 5760.426,E2 5760.426} C_VEL
LIN {X 0,Y 342.495,Z 1105.641,A -85,B 0,C 180,E1 5759.622,E2 5759.622} C_VEL
LIN {X 0,Y 327.58,Z 1123.084,A -85,B 0,C 180,E1 5758.655,E2 5758.655} C_VEL
LIN {X 0,Y 308.347,Z 1143.393,A -85,B 0,C 180,E1 5757.254,E2 5757.254} C_VEL
LIN {X 0,Y 289.809,Z 1160.776,A -85,B 0,C 180,E1 5755.709,E2 5755.709} C_VEL
LIN {X 0,Y 273.236,Z 1174.981,A -85,B 0,C 180,E1 5754.119,E2 5754.119} C_VEL
LIN {X 0,Y 256.345,Z 1188.271,A -85,B 0,C 180,E1 5752.249,E2 5752.249} C_VEL
LIN {X 0,Y 237.681,Z 1201.736,A -85,B 0,C 180,E1 5749.823,E2 5749.823} C_VEL
LIN {X 0,Y 214.304,Z 1216.934,A -85,B 0,C 180,E1 5746.08,E2 5746.08} C_VEL
LIN {X 0,Y 195.331,Z 1228.056,A -85,B 0,C 180,E1 5742.232,E2 5742.232} C_VEL
LIN {X 0,Y 178.612,Z 1237.115,A -85,B 0,C 180,E1 5737.971,E2 5737.971} C_VEL
LIN {X 0,Y 161.496,Z 1245.765,A -85,B 0,C 180,E1 5732.326,E2 5732.326} C_VEL
LIN {X 0,Y 142.047,Z 1254.907,A -85,B 0,C 180,E1 5723.25,E2 5723.25} C_VEL
LIN {X 0,Y 129.68,Z 1260.526,A -85,B 0,C 180,E1 5714.584,E2 5714.584} C_VEL
LIN {X 0,Y 120.995,Z 1264.601,A -85,B 0,C 180,E1 5705.367,E2 5705.367} C_VEL
LIN {X 0,Y 115.482,Z 1267.503,A -85,B 0,C 180,E1 5695.677,E2 5695.677} C_VEL
LIN {X 0,Y 112.662,Z 1269.458,A -85,B 0,C 180,E1 5685.465,E2 5685.465} C_VEL
LIN {X 0,Y 112.064,Z 1270.38,A -85,B 0,C 180,E1 5676.684,E2 5676.684} C_VEL
LIN {X 0,Y 112.053,Z 1270.674,A -85,B 0,C 180,E1 5669.512,E2 5669.512} C_VEL
LIN {X 0,Y 112.065,Z 1270.297,A -85,B 0,C 180,E1 5661.817,E2 5661.817} C_VEL
LIN {X 0,Y 113.333,Z 1268.927,A -85,B 0,C 180,E1 5650.973,E2 5650.973} C_VEL
LIN {X 0,Y 118.719,Z 1265.765,A -85,B 0,C 180,E1 5637.982,E2 5637.982} C_VEL
LIN {X 0,Y 127.763,Z 1261.37,A -85,B 0,C 180,E1 5627.119,E2 5627.119} C_VEL
LIN {X 0,Y 139.156,Z 1256.146,A -85,B 0,C 180,E1 5618.479,E2 5618.479} C_VEL
LIN {X 0,Y 152.342,Z 1250.041,A -85,B 0,C 180,E1 5611.472,E2 5611.472} C_VEL
LIN {X 0,Y 169.905,Z 1241.547,A -85,B 0,C 180,E1 5604.698,E2 5604.698} C_VEL
LIN {X 0,Y 191.079,Z 1230.35,A -85,B 0,C 180,E1 5598.764,E2 5598.764} C_VEL
LIN {X 0,Y 208.958,Z 1220.027,A -85,B 0,C 180,E1 5594.913,E2 5594.913} C_VEL
LIN {X 0,Y 225.818,Z 1209.492,A -85,B 0,C 180,E1 5591.959,E2 5591.959} C_VEL
LIN {X 0,Y 243.188,Z 1197.718,A -85,B 0,C 180,E1 5589.413,E2 5589.413} C_VEL
LIN {X 0,Y 263.816,Z 1182.459,A -85,B 0,C 180,E1 5586.892,E2 5586.892} C_VEL
LIN {X 0,Y 284.88,Z 1164.917,A -85,B 0,C 180,E1 5584.739,E2 5584.739} C_VEL
LIN {X 0,Y 301.399,Z 1149.793,A -85,B 0,C 180,E1 5583.288,E2 5583.288} C_VEL
LIN {X 0,Y 317.107,Z 1134.078,A -85,B 0,C 180,E1 5582.065,E2 5582.065} C_VEL
LIN {X 0,Y 333.391,Z 1116.206,A -85,B 0,C 180,E1 5580.945,E2 5580.945} C_VEL
LIN {X 0,Y 352.397,Z 1092.735,A -85,B 0,C 180,E1 5579.787,E2 5579.787} C_VEL
LIN {X 0,Y 356.806,Z 1086.805,A -85,B 0,C 180,E1 5579.528,E2 5579.528} C_VEL
LIN {X 0,Y 342.991,Z 1104.455,A -85,B 0,C 180,E1 5578.65,E2 5578.65} C_VEL
LIN {X 0,Y 329.163,Z 1120.522,A -85,B 0,C 180,E1 5577.704,E2 5577.704} C_VEL
LIN {X 0,Y 312.991,Z 1137.622,A -85,B 0,C 180,E1 5576.484,E2 5576.484} C_VEL
LIN {X 0,Y 291.195,Z 1158.16,A -85,B 0,C 180,E1 5574.606,E2 5574.606} C_VEL
LIN {X 0,Y 273.707,Z 1172.891,A -85,B 0,C 180,E1 5572.865,E2 5572.865} C_VEL
LIN {X 0,Y 257.099,Z 1185.68,A -85,B 0,C 180,E1 5570.968,E2 5570.968} C_VEL
LIN {X 0,Y 239.598,Z 1198.019,A -85,B 0,C 180,E1 5568.652,E2 5568.652} C_VEL
LIN {X 0,Y 218.129,Z 1211.783,A -85,B 0,C 180,E1 5565.227,E2 5565.227} C_VEL
LIN {X 0,Y 197.36,Z 1223.562,A -85,B 0,C 180,E1 5561.08,E2 5561.08} C_VEL
LIN {X 0,Y 180.503,Z 1232.326,A -85,B 0,C 180,E1 5556.815,E2 5556.815} C_VEL
LIN {X 0,Y 163.873,Z 1240.309,A -85,B 0,C 180,E1 5551.438,E2 5551.438} C_VEL
LIN {X 0,Y 145.092,Z 1248.644,A -85,B 0,C 180,E1 5543.039,E2 5543.039} C_VEL
LIN {X 0,Y 131.758,Z 1254.151,A -85,B 0,C 180,E1 5534.249,E2 5534.249} C_VEL
LIN {X 0,Y 122.71,Z 1257.885,A -85,B 0,C 180,E1 5525.319,E2 5525.319} C_VEL
LIN {X 0,Y 116.71,Z 1260.504,A -85,B 0,C 180,E1 5515.882,E2 5515.882} C_VEL
LIN {X 0,Y 113.323,Z 1262.234,A -85,B 0,C 180,E1 5505.849,E2 5505.849} C_VEL
LIN {X 0,Y 112.213,Z 1263.063,A -85,B 0,C 180,E1 5496.628,E2 5496.628} C_VEL
LIN {X 0,Y 112.072,Z 1263.278,A -85,B 0,C 180,E1 5488.443,E2 5488.443} C_VEL
LIN {X 0,Y 112.462,Z 1262.935,A -85,B 0,C 180,E1 5479.734,E2 5479.734} C_VEL
LIN {X 0,Y 115.027,Z 1261.39,A -85,B 0,C 180,E1 5468.028,E2 5468.028} C_VEL
LIN {X 0,Y 121.288,Z 1258.536,A -85,B 0,C 180,E1 5456.448,E2 5456.448} C_VEL
LIN {X 0,Y 130.289,Z 1254.8,A -85,B 0,C 180,E1 5446.896,E2 5446.896} C_VEL
LIN {X 0,Y 141.473,Z 1250.178,A -85,B 0,C 180,E1 5438.947,E2 5438.947} C_VEL
LIN {X 0,Y 155.528,Z 1244.15,A -85,B 0,C 180,E1 5431.815,E2 5431.815} C_VEL
LIN {X 0,Y 175.061,Z 1235.19,A -85,B 0,C 180,E1 5424.72,E2 5424.72} C_VEL
LIN {X 0,Y 194.285,Z 1225.329,A -85,B 0,C 180,E1 5419.544,E2 5419.544} C_VEL
LIN {X 0,Y 211.408,Z 1215.786,A -85,B 0,C 180,E1 5415.922,E2 5415.922} C_VEL
LIN {X 0,Y 228.917,Z 1205.148,A -85,B 0,C 180,E1 5412.872,E2 5412.872} C_VEL
LIN {X 0,Y 250.634,Z 1190.665,A -85,B 0,C 180,E1 5409.764,E2 5409.764} C_VEL
LIN {X 0,Y 271.211,Z 1175.102,A -85,B 0,C 180,E1 5407.321,E2 5407.321} C_VEL
LIN {X 0,Y 287.405,Z 1161.683,A -85,B 0,C 180,E1 5405.673,E2 5405.673} C_VEL
LIN {X 0,Y 303.81,Z 1146.82,A -85,B 0,C 180,E1 5404.199,E2 5404.199} C_VEL
LIN {X 0,Y 320.498,Z 1130.222,A -85,B 0,C 180,E1 5402.861,E2 5402.861} C_VEL
LIN {X 0,Y 340.099,Z 1108.327,A -85,B 0,C 180,E1 5401.463,E2 5401.463} C_VEL
LIN {X 0,Y 354.501,Z 1090.263,A -85,B 0,C 180,E1 5400.534,E2 5400.534} C_VEL
LIN {X 0,Y 356.276,Z 1087.907,A -85,B 0,C 180,E1 5400.426,E2 5400.426} C_VEL
LIN {X 0,Y 349.506,Z 1096.978,A -85,B 0,C 180,E1 5400.193,E2 5400.193} C_VEL
LIN {X 0,Y 341.444,Z 1106.794,A -85,B 0,C 180,E1 5400.242,E2 5400.242} C_VEL
LIN {X 0,Y 332.195,Z 1117.544,A -85,B 0,C 180,E1 5400.61,E2 5400.61} C_VEL
LIN {X 0,Y 325.823,Z 1124.556,A -85,B 0,C 180,E1 5401.006,E2 5401.006} C_VEL
LIN {X 0,Y 305.283,Z 1145.26,A -85,B 0,C 180,E1 5402.493,E2 5402.493} C_VEL
LIN {X 0,Y 288.651,Z 1160.285,A -85,B 0,C 180,E1 5403.859,E2 5403.859} C_VEL
LIN {X 0,Y 272.204,Z 1173.853,A -85,B 0,C 180,E1 5405.391,E2 5405.391} C_VEL
LIN {X 0,Y 255.026,Z 1186.803,A -85,B 0,C 180,E1 5407.222,E2 5407.222} C_VEL
LIN {X 0,Y 233.507,Z 1201.554,A -85,B 0,C 180,E1 5409.933,E2 5409.933} C_VEL
LIN {X 0,Y 211.691,Z 1214.693,A -85,B 0,C 180,E1 5413.303,E2 5413.303} C_VEL
LIN {X 0,Y 193.293,Z 1224.745,A -85,B 0,C 180,E1 5416.839,E2 5416.839} C_VEL
LIN {X 0,Y 175.753,Z 1233.493,A -85,B 0,C 180,E1 5421.056,E2 5421.056} C_VEL
LIN {X 0,Y 155.571,Z 1242.708,A -85,B 0,C 180,E1 5427.477,E2 5427.477} C_VEL
LIN {X 0,Y 137.654,Z 1249.962,A -85,B 0,C 180,E1 5435.528,E2 5435.528} C_VEL
LIN {X 0,Y 124.879,Z 1254.875,A -85,B 0,C 180,E1 5443.868,E2 5443.868} C_VEL
LIN {X 0,Y 115.267,Z 1258.504,A -85,B 0,C 180,E1 5453.209,E2 5453.209} C_VEL
LIN {X 0,Y 108.622,Z 1261.125,A -85,B 0,C 180,E1 5463.753,E2 5463.753} C_VEL
LIN {X 0,Y 105.183,Z 1262.708,A -85,B 0,C 180,E1 5474.538,E2 5474.538} C_VEL
LIN {X 0,Y 104.212,Z 1263.353,A -85,B 0,C 180,E1 5483.364,E2 5483.364} C_VEL
LIN {X 0,Y 104.079,Z 1263.534,A -85,B 0,C 180,E1 5491.626,E2 5491.626} C_VEL
LIN {X 0,Y 104.54,Z 1263.188,A -85,B 0,C 180,E1 5501.002,E2 5501.002} C_VEL
LIN {X 0,Y 107.506,Z 1261.625,A -85,B 0,C 180,E1 5513.546,E2 5513.546} C_VEL
LIN {X 0,Y 114.525,Z 1258.76,A -85,B 0,C 180,E1 5525.77,E2 5525.77} C_VEL
LIN {X 0,Y 124.381,Z 1255.015,A -85,B 0,C 180,E1 5535.648,E2 5535.648} C_VEL
LIN {X 0,Y 137.041,Z 1250.138,A -85,B 0,C 180,E1 5544.048,E2 5544.048} C_VEL
LIN {X 0,Y 154.111,Z 1243.211,A -85,B 0,C 180,E1 5551.889,E2 5551.889} C_VEL
LIN {X 0,Y 174.946,Z 1233.783,A -85,B 0,C 180,E1 5558.638,E2 5558.638} C_VEL
LIN {X 0,Y 192.435,Z 1225.078,A -85,B 0,C 180,E1 5562.895,E2 5562.895} C_VEL
LIN {X 0,Y 209.89,Z 1215.581,A -85,B 0,C 180,E1 5566.301,E2 5566.301} C_VEL
LIN {X 0,Y 228.869,Z 1204.254,A -85,B 0,C 180,E1 5569.336,E2 5569.336} C_VEL
LIN {X 0,Y 252.147,Z 1188.709,A -85,B 0,C 180,E1 5572.366,E2 5572.366} C_VEL
LIN {X 0,Y 270.23,Z 1175.197,A -85,B 0,C 180,E1 5574.333,E2 5574.333} C_VEL
LIN {X 0,Y 286.645,Z 1161.766,A -85,B 0,C 180,E1 5575.885,E2 5575.885} C_VEL
LIN {X 0,Y 302.266,Z 1147.803,A -85,B 0,C 180,E1 5577.191,E2 5577.191} C_VEL
LIN {X 0,Y 318.067,Z 1132.347,A -85,B 0,C 180,E1 5578.379,E2 5578.379} C_VEL
LIN {X 0,Y 334.036,Z 1115.171,A -85,B 0,C 180,E1 5579.482,E2 5579.482} C_VEL
LIN {X 0,Y 317.291,Z 1133.417,A -85,B 0,C 180,E1 5580.542,E2 5580.542} C_VEL
LIN {X 0,Y 301.531,Z 1149.049,A -85,B 0,C 180,E1 5581.67,E2 5581.67} C_VEL
LIN {X 0,Y 285.29,Z 1163.783,A -85,B 0,C 180,E1 5582.973,E2 5582.973} C_VEL
LIN {X 0,Y 264.868,Z 1180.678,A -85,B 0,C 180,E1 5584.877,E2 5584.877} C_VEL
LIN {X 0,Y 242.849,Z 1196.825,A -85,B 0,C 180,E1 5587.333,E2 5587.333} C_VEL
LIN {X 0,Y 224.22,Z 1209.213,A -85,B 0,C 180,E1 5589.847,E2 5589.847} C_VEL
LIN {X 0,Y 206.05,Z 1220.275,A -85,B 0,C 180,E1 5592.812,E2 5592.812} C_VEL
LIN {X 0,Y 184.271,Z 1232.42,A -85,B 0,C 180,E1 5597.311,E2 5597.311} C_VEL
LIN {X 0,Y 163.058,Z 1242.886,A -85,B 0,C 180,E1 5603.149,E2 5603.149} C_VEL
LIN {X 0,Y 147.397,Z 1250.077,A -85,B 0,C 180,E1 5608.987,E2 5608.987} C_VEL
LIN {X 0,Y 133.466,Z 1256.134,A -85,B 0,C 180,E1 5616.03,E2 5616.03} C_VEL
LIN {X 0,Y 120.782,Z 1261.527,A -85,B 0,C 180,E1 5625.312,E2 5625.312} C_VEL
LIN {X 0,Y 109.912,Z 1266.363,A -85,B 0,C 180,E1 5638.795,E2 5638.795} C_VEL
LIN {X 0,Y 105.239,Z 1268.883,A -85,B 0,C 180,E1 5651.181,E2 5651.181} C_VEL
LIN {X 0,Y 104.07,Z 1270.059,A -85,B 0,C 180,E1 5661.74,E2 5661.74} C_VEL
LIN {X 0,Y 104.058,Z 1270.411,A -85,B 0,C 180,E1 5669.475,E2 5669.475} C_VEL
LIN {X 0,Y 104.072,Z 1270.115,A -85,B 0,C 180,E1 5677.2,E2 5677.2} C_VEL
LIN {X 0,Y 104.922,Z 1269.116,A -85,B 0,C 180,E1 5687.208,E2 5687.208} C_VEL
LIN {X 0,Y 108.34,Z 1267.11,A -85,B 0,C 180,E1 5698.104,E2 5698.104} C_VEL
LIN {X 0,Y 115.108,Z 1263.99,A -85,B 0,C 180,E1 5708.74,E2 5708.74} C_VEL
LIN {X 0,Y 126.539,Z 1259.167,A -85,B 0,C 180,E1 5719.367,E2 5719.367} C_VEL
LIN {X 0,Y 144.254,Z 1251.563,A -85,B 0,C 180,E1 5729.602,E2 5729.602} C_VEL
LIN {X 0,Y 160.807,Z 1244.03,A -85,B 0,C 180,E1 5736.102,E2 5736.102} C_VEL
LIN {X 0,Y 177.633,Z 1235.819,A -85,B 0,C 180,E1 5741.062,E2 5741.062} C_VEL
LIN {X 0,Y 196.406,Z 1225.897,A -85,B 0,C 180,E1 5745.341,E2 5745.341} C_VEL
LIN {X 0,Y 220.633,Z 1211.638,A -85,B 0,C 180,E1 5749.6,E2 5749.6} C_VEL
